LIN {X 0,Y 291.384,Z 318.187,A -85,B 0,C 180,E1 -16597.255,E2 -16597.255} C_VEL
LIN {X 0,Y 291.337,Z 318.196,A -85,B 0,C 180,E1 -16600.642,E2 -16600.642} C_VEL
LIN {X 0,Y 291.402,Z 318.333,A -85,B 0,C 180,E1 -16602.352,E2 -16602.352} C_VEL
LIN {X 0,Y 292.391,Z 323.725,A -85,B 0,C 180,E1 -16606.145,E2 -16606.145} C_VEL
LIN {X 0,Y 293.452,Z 329.609,A -85,B 0,C 180,E1 -16610.03,E2 -16610.03} C_VEL
LIN {X 0,Y 293.964,Z 332.856,A -85,B 0,C 180,E1 -16612.088,E2 -16612.088} C_VEL
LIN {X 0,Y 294.034,Z 334.839,A -85,B 0,C 180,E1 -16613.305,E2 -16613.305} C_VEL
LIN {X 0,Y 293.395,Z 338.972,A -85,B 0,C 180,E1 -16615.742,E2 -16615.742} C_VEL
LIN {X 0,Y 292.231,Z 346.349,A -85,B 0,C 180,E1 -16619.972,E2 -16619.972} C_VEL
LIN {X 0,Y 291.163,Z 353.918,A -85,B 0,C 180,E1 -16624.248,E2 -16624.248} C_VEL
LIN {X 0,Y 290.715,Z 358.235,A -85,B 0,C 180,E1 -16626.649,E2 -16626.649} C_VEL
LIN {X 0,Y 292.536,Z 371.557,A -85,B 0,C 180,E1 -16627.394,E2 -16627.394} C_VEL
LIN {X 0,Y 293.951,Z 383.978,A -85,B 0,C 180,E1 -16628.327,E2 -16628.327} C_VEL
LIN {X 0,Y 294.913,Z 395.491,A -85,B 0,C 180,E1 -16629.421,E2 -16629.421} C_VEL
LIN {X 0,Y 295.433,Z 406.744,A -85,B 0,C 180,E1 -16630.727,E2 -16630.727} C_VEL
LIN {X 0,Y 294.037,Z 417.883,A -85,B 0,C 180,E1 -16632.257,E2 -16632.257} C_VEL
LIN {X 0,Y 292.817,Z 426.678,A -85,B 0,C 180,E1 -16633.752,E2 -16633.752} C_VEL
LIN {X 0,Y 291.678,Z 435.982,A -85,B 0,C 180,E1 -16635.701,E2 -16635.701} C_VEL
LIN {X 0,Y 290.738,Z 444.013,A -85,B 0,C 180,E1 -16637.789,E2 -16637.789} C_VEL
LIN {X 0,Y 290.233,Z 449.451,A -85,B 0,C 180,E1 -16639.536,E2 -16639.536} C_VEL
LIN {X 0,Y 289.879,Z 454.755,A -85,B 0,C 180,E1 -16641.636,E2 -16641.636} C_VEL
LIN {X 0,Y 289.804,Z 459.093,A -85,B 0,C 180,E1 -16643.875,E2 -16643.875} C_VEL
LIN {X 0,Y 289.76,Z 461.832,A -85,B 0,C 180,E1 -16645.827,E2 -16645.827} C_VEL
LIN {X 0,Y 289.832,Z 463.266,A -85,B 0,C 180,E1 -16647.22,E2 -16647.22} C_VEL
LIN {X 0,Y 290.028,Z 464.247,A -85,B 0,C 180,E1 -16648.611,E2 -16648.611} C_VEL
LIN {X 0,Y 290.042,Z 464.802,A -85,B 0,C 180,E1 -16650,E2 -16650} C_VEL
LIN {X 0,Y 289.962,Z 464.944,A -85,B 0,C 180,E1 -16651.389,E2 -16651.389} C_VEL
LIN {X 0,Y 289.747,Z 464.648,A -85,B 0,C 180,E1 -16652.781,E2 -16652.781} C_VEL
LIN {X 0,Y 289.673,Z 463.929,A -85,B 0,C 180,E1 -16654.174,E2 -16654.174} C_VEL
LIN {X 0,Y 289.656,Z 461.291,A -85,B 0,C 180,E1 -16656.968,E2 -16656.968} C_VEL
LIN {X 0,Y 289.897,Z 458.175,A -85,B 0,C 180,E1 -16659.067,E2 -16659.067} C_VEL
LIN {X 0,Y 290.384,Z 454.047,A -85,B 0,C 180,E1 -16661.164,E2 -16661.164} C_VEL
LIN {X 0,Y 291.558,Z 447.849,A -85,B 0,C 180,E1 -16663.593,E2 -16663.593} C_VEL
LIN {X 0,Y 292.919,Z 441.128,A -85,B 0,C 180,E1 -16665.66,E2 -16665.66} C_VEL
LIN {X 0,Y 294.474,Z 433.033,A -85,B 0,C 180,E1 -16667.68,E2 -16667.68} C_VEL
LIN {X 0,Y 296.368,Z 424.574,A -85,B 0,C 180,E1 -16669.39,E2 -16669.39} C_VEL
LIN {X 0,Y 298.591,Z 414.589,A -85,B 0,C 180,E1 -16671.035,E2 -16671.035} C_VEL
LIN {X 0,Y 299.453,Z 405.428,A -85,B 0,C 180,E1 -16672.367,E2 -16672.367} C_VEL
LIN {X 0,Y 299.529,Z 394.395,A -85,B 0,C 180,E1 -16673.783,E2 -16673.783} C_VEL
LIN {X 0,Y 298.6,Z 383.187,A -85,B 0,C 180,E1 -16675.066,E2 -16675.066} C_VEL
LIN {X 0,Y 296.529,Z 370.803,A -85,B 0,C 180,E1 -16676.361,E2 -16676.361} C_VEL
LIN {X 0,Y 293.021,Z 357.071,A -85,B 0,C 180,E1 -16677.694,E2 -16677.694} C_VEL
LIN {X 0,Y 291.962,Z 353.125,A -85,B 0,C 180,E1 -16678.074,E2 -16678.074} C_VEL
LIN {X 0,Y 293.008,Z 346.862,A -85,B 0,C 180,E1 -16681.849,E2 -16681.849} C_VEL
LIN {X 0,Y 294.347,Z 340.748,A -85,B 0,C 180,E1 -16685.727,E2 -16685.727} C_VEL
LIN {X 0,Y 294.85,Z 338.347,A -85,B 0,C 180,E1 -16687.329,E2 -16687.329} C_VEL
LIN {X 0,Y 294.381,Z 334.557,A -85,B 0,C 180,E1 -16690.185,E2 -16690.185} C_VEL
LIN {X 0,Y 293.552,Z 329.912,A -85,B 0,C 180,E1 -16694.09,E2 -16694.09} C_VEL
LIN {X 0,Y 292.79,Z 325.8,A -85,B 0,C 180,E1 -16698.083,E2 -16698.083} C_VEL
LIN {X 0,Y 292.287,Z 322.897,A -85,B 0,C 180,E1 -16701.305,E2 -16701.305} C_VEL
LIN {X 0,Y 291.735,Z 320.101,A -85,B 0,C 180,E1 -16704.993,E2 -16704.993} C_VEL
LIN {X 0,Y 291.376,Z 318.246,A -85,B 0,C 180,E1 -16707.951,E2 -16707.951} C_VEL
LIN {X 0,Y 291.386,Z 318.19,A -85,B 0,C 180,E1 -16711.158,E2 -16711.158} C_VEL
LIN {X 0,Y 291.421,Z 318.185,A -85,B 0,C 180,E1 -16714.272,E2 -16714.272} C_VEL
LIN {X 0,Y 291.386,Z 318.187,A -85,B 0,C 180,E1 -16717.3,E2 -16717.3} C_VEL
LIN {X 0,Y 291.463,Z 318.177,A -85,B 0,C 180,E1 -16720.27,E2 -16720.27} C_VEL
LIN {X 0,Y 291.559,Z 318.164,A -85,B 0,C 180,E1 -16724.624,E2 -16724.624} C_VEL
LIN {X 0,Y 291.533,Z 318.167,A -85,B 0,C 180,E1 -16728.88,E2 -16728.88} C_VEL
LIN {X 0,Y 291.667,Z 318.152,A -85,B 0,C 180,E1 -16731.687,E2 -16731.687} C_VEL
LIN {X 0,Y 291.615,Z 318.162,A -85,B 0,C 180,E1 -16734.468,E2 -16734.468} C_VEL
LIN {X 0,Y 291.892,Z 318.126,A -85,B 0,C 180,E1 -16738.62,E2 -16738.62} C_VEL
LIN {X 0,Y 291.893,Z 318.128,A -85,B 0,C 180,E1 -16741.379,E2 -16741.379} C_VEL
LIN {X 0,Y 291.907,Z 319.951,A -85,B 0,C 180,E1 -16745.526,E2 -16745.526} C_VEL
LIN {X 0,Y 292.082,Z 321.378,A -85,B 0,C 180,E1 -16748.301,E2 -16748.301} C_VEL
LIN {X 0,Y 291.958,Z 322.586,A -85,B 0,C 180,E1 -16750.134,E2 -16750.134} C_VEL
LIN {X 0,Y 293.139,Z 325.506,A -85,B 0,C 180,E1 -16750.48,E2 -16750.48} C_VEL
LIN {X 0,Y 296.261,Z 331.803,A -85,B 0,C 180,E1 -16751.329,E2 -16751.329} C_VEL
LIN {X 0,Y 300.206,Z 341.684,A -85,B 0,C 180,E1 -16752.657,E2 -16752.657} C_VEL
LIN {X 0,Y 303.281,Z 352.214,A -85,B 0,C 180,E1 -16754.103,E2 -16754.103} C_VEL
LIN {X 0,Y 304.6,Z 358.809,A -85,B 0,C 180,E1 -16755.044,E2 -16755.044} C_VEL
LIN {X 0,Y 302.617,Z 370.426,A -85,B 0,C 180,E1 -16756.462,E2 -16756.462} C_VEL
LIN {X 0,Y 300.635,Z 380.69,A -85,B 0,C 180,E1 -16758.044,E2 -16758.044} C_VEL
LIN {X 0,Y 298.697,Z 389.576,A -85,B 0,C 180,E1 -16759.752,E2 -16759.752} C_VEL
LIN {X 0,Y 296.547,Z 398.595,A -85,B 0,C 180,E1 -16761.91,E2 -16761.91} C_VEL
LIN {X 0,Y 294.907,Z 405.165,A -85,B 0,C 180,E1 -16763.899,E2 -16763.899} C_VEL
LIN {X 0,Y 293.27,Z 411.348,A -85,B 0,C 180,E1 -16766.317,E2 -16766.317} C_VEL
LIN {X 0,Y 292.017,Z 416.012,A -85,B 0,C 180,E1 -16768.773,E2 -16768.773} C_VEL
LIN {X 0,Y 291.311,Z 418.312,A -85,B 0,C 180,E1 -16770.44,E2 -16770.44} C_VEL
LIN {X 0,Y 290.723,Z 420.115,A -85,B 0,C 180,E1 -16772.21,E2 -16772.21} C_VEL
LIN {X 0,Y 290.166,Z 421.443,A -85,B 0,C 180,E1 -16774.563,E2 -16774.563} C_VEL
LIN {X 0,Y 289.816,Z 421.556,A -85,B 0,C 180,E1 -16777.319,E2 -16777.319} C_VEL
LIN {X 0,Y 289.773,Z 420.803,A -85,B 0,C 180,E1 -16779.094,E2 -16779.094} C_VEL
LIN {X 0,Y 289.911,Z 418.967,A -85,B 0,C 180,E1 -16781.279,E2 -16781.279} C_VEL
LIN {X 0,Y 290.27,Z 416.159,A -85,B 0,C 180,E1 -16783.418,E2 -16783.418} C_VEL
LIN {X 0,Y 290.82,Z 411.521,A -85,B 0,C 180,E1 -16785.913,E2 -16785.913} C_VEL
LIN {X 0,Y 291.592,Z 405.427,A -85,B 0,C 180,E1 -16788.346,E2 -16788.346} C_VEL
LIN {X 0,Y 292.521,Z 398.224,A -85,B 0,C 180,E1 -16790.564,E2 -16790.564} C_VEL
LIN {X 0,Y 293.568,Z 390.435,A -85,B 0,C 180,E1 -16792.494,E2 -16792.494} C_VEL
LIN {X 0,Y 294.849,Z 381.177,A -85,B 0,C 180,E1 -16794.356,E2 -16794.356} C_VEL
LIN {X 0,Y 296.27,Z 370.145,A -85,B 0,C 180,E1 -16796.125,E2 -16796.125} C_VEL
LIN {X 0,Y 297.43,Z 359.208,A -85,B 0,C 180,E1 -16797.539,E2 -16797.539} C_VEL
LIN {X 0,Y 298.285,Z 349.136,A -85,B 0,C 180,E1 -16798.589,E2 -16798.589} C_VEL
LIN {X 0,Y 295.879,Z 337.582,A -85,B 0,C 180,E1 -16799.734,E2 -16799.734} C_VEL
LIN {X 0,Y 292.465,Z 324.071,A -85,B 0,C 180,E1 -16800.819,E2 -16800.819} C_VEL
LIN {X 0,Y 290.677,Z 318.279,A -85,B 0,C 180,E1 -16801.23,E2 -16801.23} C_VEL
LIN {X 0,Y 291.025,Z 318.232,A -85,B 0,C 180,E1 -16804.235,E2 -16804.235} C_VEL
LIN {X 0,Y 291.29,Z 318.203,A -85,B 0,C 180,E1 -16807.292,E2 -16807.292} C_VEL
LIN {X 0,Y 291.385,Z 318.187,A -85,B 0,C 180,E1 -16810.265,E2 -16810.265} C_VEL
LIN {X 0,Y 291.498,Z 318.174,A -85,B 0,C 180,E1 -16814.665,E2 -16814.665} C_VEL
LIN {X 0,Y 291.536,Z 318.172,A -85,B 0,C 180,E1 -16818.88,E2 -16818.88} C_VEL
LIN {X 0,Y 291.655,Z 318.154,A -85,B 0,C 180,E1 -16821.687,E2 -16821.687} C_VEL
LIN {X 0,Y 291.612,Z 318.159,A -85,B 0,C 180,E1 -16824.468,E2 -16824.468} C_VEL
LIN {X 0,Y 291.89,Z 318.127,A -85,B 0,C 180,E1 -16828.62,E2 -16828.62} C_VEL
LIN {X 0,Y 291.889,Z 318.123,A -85,B 0,C 180,E1 -16831.38,E2 -16831.38} C_VEL
LIN {X 0,Y 291.613,Z 318.158,A -85,B 0,C 180,E1 -16835.532,E2 -16835.532} C_VEL
LIN {X 0,Y 291.669,Z 318.153,A -85,B 0,C 180,E1 -16838.913,E2 -16838.913} C_VEL
LIN {X 0,Y 291.521,Z 318.174,A -85,B 0,C 180,E1 -16842.531,E2 -16842.531} C_VEL
LIN {X 0,Y 291.556,Z 318.164,A -85,B 0,C 180,E1 -16845.376,E2 -16845.376} C_VEL
LIN {X 0,Y 291.451,Z 318.179,A -85,B 0,C 180,E1 -16849.875,E2 -16849.875} C_VEL
LIN {X 0,Y 291.401,Z 318.188,A -85,B 0,C 180,E1 -16854.205,E2 -16854.205} C_VEL
LIN {X 0,Y 291.424,Z 318.181,A -85,B 0,C 180,E1 -16857.272,E2 -16857.272} C_VEL
LIN {X 0,Y 291.338,Z 318.194,A -85,B 0,C 180,E1 -16860.437,E2 -16860.437} C_VEL
LIN {X 0,Y 291.346,Z 318.193,A -85,B 0,C 180,E1 -16863.699,E2 -16863.699} C_VEL
LIN {X 0,Y 291.385,Z 318.186,A -85,B 0,C 180,E1 -16867.256,E2 -16867.256} C_VEL
LIN {X 0,Y 291.335,Z 318.193,A -85,B 0,C 180,E1 -16870.643,E2 -16870.643} C_VEL
LIN {X 0,Y 291.291,Z 318.198,A -85,B 0,C 180,E1 -16874.402,E2 -16874.402} C_VEL
LIN {X 0,Y 291.328,Z 318.194,A -85,B 0,C 180,E1 -16878.405,E2 -16878.405} C_VEL
LIN {X 0,Y 291.366,Z 318.19,A -85,B 0,C 180,E1 -16881.16,E2 -16881.16} C_VEL
LIN {X 0,Y 291.363,Z 318.188,A -85,B 0,C 180,E1 -16884.626,E2 -16884.626} C_VEL
LIN {X 0,Y 291.374,Z 318.189,A -85,B 0,C 180,E1 -16887.951,E2 -16887.951} C_VEL
LIN {X 0,Y 291.388,Z 318.188,A -85,B 0,C 180,E1 -16891.159,E2 -16891.159} C_VEL
LIN {X 0,Y 291.422,Z 318.181,A -85,B 0,C 180,E1 -16894.273,E2 -16894.273} C_VEL
LIN {X 0,Y 291.375,Z 318.192,A -85,B 0,C 180,E1 -16897.299,E2 -16897.299} C_VEL
LIN {X 0,Y 291.442,Z 318.178,A -85,B 0,C 180,E1 -16900.269,E2 -16900.269} C_VEL
LIN {X 0,Y 291.5,Z 318.173,A -85,B 0,C 180,E1 -16904.665,E2 -16904.665} C_VEL
LIN {X 0,Y 291.533,Z 318.17,A -85,B 0,C 180,E1 -16908.881,E2 -16908.881} C_VEL
LIN {X 0,Y 291.671,Z 318.151,A -85,B 0,C 180,E1 -16911.688,E2 -16911.688} C_VEL
LIN {X 0,Y 291.626,Z 318.157,A -85,B 0,C 180,E1 -16914.468,E2 -16914.468} C_VEL
LIN {X 0,Y 291.89,Z 318.125,A -85,B 0,C 180,E1 -16918.621,E2 -16918.621} C_VEL
LIN {X 0,Y 291.867,Z 318.126,A -85,B 0,C 180,E1 -16921.547,E2 -16921.547} C_VEL
LIN {X 0,Y 291.099,Z 318.226,A -85,B 0,C 180,E1 -16922.696,E2 -16922.696} C_VEL
LIN {X 0,Y 288.184,Z 318.588,A -85,B 0,C 180,E1 -16924.567,E2 -16924.567} C_VEL
LIN {X 0,Y 285.759,Z 318.889,A -85,B 0,C 180,E1 -16926.085,E2 -16926.085} C_VEL
LIN {X 0,Y 284.709,Z 319.019,A -85,B 0,C 180,E1 -16927.262,E2 -16927.262} C_VEL
LIN {X 0,Y 284.616,Z 319.029,A -85,B 0,C 180,E1 -16927.661,E2 -16927.661} C_VEL
LIN {X 0,Y 284.486,Z 319.046,A -85,B 0,C 180,E1 -16931.399,E2 -16931.399} C_VEL
LIN {X 0,Y 284.451,Z 319.05,A -85,B 0,C 180,E1 -16935.508,E2 -16935.508} C_VEL
LIN {X 0,Y 284.371,Z 319.063,A -85,B 0,C 180,E1 -16940.243,E2 -16940.243} C_VEL
LIN {X 0,Y 284.329,Z 319.064,A -85,B 0,C 180,E1 -16943.855,E2 -16943.855} C_VEL
LIN {X 0,Y 284.294,Z 319.068,A -85,B 0,C 180,E1 -16948.015,E2 -16948.015} C_VEL
LIN {X 0,Y 284.29,Z 319.07,A -85,B 0,C 180,E1 -16951.275,E2 -16951.275} C_VEL
LIN {X 0,Y 284.344,Z 319.064,A -85,B 0,C 180,E1 -16955.348,E2 -16955.348} C_VEL
LIN {X 0,Y 284.321,Z 319.071,A -85,B 0,C 180,E1 -16958.168,E2 -16958.168} C_VEL
LIN {X 0,Y 284.352,Z 319.177,A -85,B 0,C 180,E1 -16962.017,E2 -16962.017} C_VEL
LIN {X 0,Y 285.255,Z 324.139,A -85,B 0,C 180,E1 -16965.602,E2 -16965.602} C_VEL
LIN {X 0,Y 286.31,Z 329.908,A -85,B 0,C 180,E1 -16969.549,E2 -16969.549} C_VEL
LIN {X 0,Y 286.927,Z 334.071,A -85,B 0,C 180,E1 -16972.24,E2 -16972.24} C_VEL
LIN {X 0,Y 286.847,Z 336.875,A -85,B 0,C 180,E1 -16973.983,E2 -16973.983} C_VEL
LIN {X 0,Y 285.62,Z 343.702,A -85,B 0,C 180,E1 -16978.06,E2 -16978.06} C_VEL
LIN {X 0,Y 284.599,Z 350.468,A -85,B 0,C 180,E1 -16982.018,E2 -16982.018} C_VEL
LIN {X 0,Y 283.704,Z 357.726,A -85,B 0,C 180,E1 -16986.181,E2 -16986.181} C_VEL
LIN {X 0,Y 285.594,Z 371.626,A -85,B 0,C 180,E1 -16987.005,E2 -16987.005} C_VEL
LIN {X 0,Y 287.068,Z 385.13,A -85,B 0,C 180,E1 -16988.078,E2 -16988.078} C_VEL
LIN {X 0,Y 287.989,Z 397.037,A -85,B 0,C 180,E1 -16989.277,E2 -16989.277} C_VEL
LIN {X 0,Y 288.397,Z 407.882,A -85,B 0,C 180,E1 -16990.608,E2 -16990.608} C_VEL
LIN {X 0,Y 286.951,Z 418.62,A -85,B 0,C 180,E1 -16992.173,E2 -16992.173} C_VEL
LIN {X 0,Y 285.492,Z 428.312,A -85,B 0,C 180,E1 -16993.922,E2 -16993.922} C_VEL
LIN {X 0,Y 284.768,Z 434.847,A -85,B 0,C 180,E1 -16995.347,E2 -16995.347} C_VEL
LIN {X 0,Y 283.767,Z 442.978,A -85,B 0,C 180,E1 -16997.484,E2 -16997.484} C_VEL
LIN {X 0,Y 283.186,Z 448.5,A -85,B 0,C 180,E1 -16999.273,E2 -16999.273} C_VEL
LIN {X 0,Y 282.836,Z 453.891,A -85,B 0,C 180,E1 -17001.426,E2 -17001.426} C_VEL
LIN {X 0,Y 282.723,Z 458.606,A -85,B 0,C 180,E1 -17003.899,E2 -17003.899} C_VEL
LIN {X 0,Y 282.695,Z 461.113,A -85,B 0,C 180,E1 -17005.723,E2 -17005.723} C_VEL
LIN {X 0,Y 282.745,Z 462.6,A -85,B 0,C 180,E1 -17007.15,E2 -17007.15} C_VEL
LIN {X 0,Y 282.966,Z 463.625,A -85,B 0,C 180,E1 -17008.577,E2 -17008.577} C_VEL
LIN {X 0,Y 282.985,Z 464.21,A -85,B 0,C 180,E1 -17010,E2 -17010} C_VEL
LIN {X 0,Y 282.883,Z 464.379,A -85,B 0,C 180,E1 -17011.424,E2 -17011.424} C_VEL
LIN {X 0,Y 282.659,Z 464.133,A -85,B 0,C 180,E1 -17012.85,E2 -17012.85} C_VEL
LIN {X 0,Y 282.58,Z 463.45,A -85,B 0,C 180,E1 -17014.279,E2 -17014.279} C_VEL
LIN {X 0,Y 282.58,Z 460.876,A -85,B 0,C 180,E1 -17017.144,E2 -17017.144} C_VEL
LIN {X 0,Y 282.854,Z 457.839,A -85,B 0,C 180,E1 -17019.294,E2 -17019.294} C_VEL
LIN {X 0,Y 283.368,Z 453.789,A -85,B 0,C 180,E1 -17021.444,E2 -17021.444} C_VEL
LIN {X 0,Y 284.421,Z 448.646,A -85,B 0,C 180,E1 -17023.577,E2 -17023.577} C_VEL
LIN {X 0,Y 285.777,Z 442.264,A -85,B 0,C 180,E1 -17025.695,E2 -17025.695} C_VEL
LIN {X 0,Y 287.383,Z 434.737,A -85,B 0,C 180,E1 -17027.726,E2 -17027.726} C_VEL
LIN {X 0,Y 289.254,Z 426.605,A -85,B 0,C 180,E1 -17029.517,E2 -17029.517} C_VEL
LIN {X 0,Y 291.765,Z 416.103,A -85,B 0,C 180,E1 -17031.367,E2 -17031.367} C_VEL
LIN {X 0,Y 292.691,Z 409.429,A -85,B 0,C 180,E1 -17032.407,E2 -17032.407} C_VEL
LIN {X 0,Y 293.122,Z 399.424,A -85,B 0,C 180,E1 -17033.818,E2 -17033.818} C_VEL
LIN {X 0,Y 292.66,Z 388.197,A -85,B 0,C 180,E1 -17035.23,E2 -17035.23} C_VEL
LIN {X 0,Y 291.003,Z 375.62,A -85,B 0,C 180,E1 -17036.672,E2 -17036.672} C_VEL
LIN {X 0,Y 288.042,Z 362.704,A -85,B 0,C 180,E1 -17038.051,E2 -17038.051} C_VEL
LIN {X 0,Y 285.786,Z 355.242,A -85,B 0,C 180,E1 -17038.832,E2 -17038.832} C_VEL
LIN {X 0,Y 285.183,Z 352.471,A -85,B 0,C 180,E1 -17039.064,E2 -17039.064} C_VEL
LIN {X 0,Y 286.522,Z 345.449,A -85,B 0,C 180,E1 -17043.49,E2 -17043.49} C_VEL
LIN {X 0,Y 287.518,Z 341.303,A -85,B 0,C 180,E1 -17046.231,E2 -17046.231} C_VEL
LIN {X 0,Y 287.848,Z 339.323,A -85,B 0,C 180,E1 -17047.618,E2 -17047.618} C_VEL
LIN {X 0,Y 287.338,Z 335.397,A -85,B 0,C 180,E1 -17050.691,E2 -17050.691} C_VEL
LIN {X 0,Y 286.526,Z 330.884,A -85,B 0,C 180,E1 -17054.657,E2 -17054.657} C_VEL
LIN {X 0,Y 285.842,Z 327.153,A -85,B 0,C 180,E1 -17058.405,E2 -17058.405} C_VEL
LIN {X 0,Y 285.283,Z 324.056,A -85,B 0,C 180,E1 -17062.03,E2 -17062.03} C_VEL
LIN {X 0,Y 284.811,Z 321.631,A -85,B 0,C 180,E1 -17065.42,E2 -17065.42} C_VEL
LIN {X 0,Y 284.398,Z 319.649,A -85,B 0,C 180,E1 -17068.738,E2 -17068.738} C_VEL
LIN {X 0,Y 284.362,Z 319.065,A -85,B 0,C 180,E1 -17070.376,E2 -17070.376} C_VEL
LIN {X 0,Y 284.382,Z 319.062,A -85,B 0,C 180,E1 -17073.587,E2 -17073.587} C_VEL
LIN {X 0,Y 284.371,Z 319.065,A -85,B 0,C 180,E1 -17076.707,E2 -17076.707} C_VEL
LIN {X 0,Y 284.409,Z 319.059,A -85,B 0,C 180,E1 -17081.262,E2 -17081.262} C_VEL
LIN {X 0,Y 284.496,Z 319.043,A -85,B 0,C 180,E1 -17084.459,E2 -17084.459} C_VEL
LIN {X 0,Y 284.487,Z 319.046,A -85,B 0,C 180,E1 -17088.601,E2 -17088.601} C_VEL
LIN {X 0,Y 284.622,Z 319.028,A -85,B 0,C 180,E1 -17091.48,E2 -17091.48} C_VEL
LIN {X 0,Y 284.584,Z 319.038,A -85,B 0,C 180,E1 -17094.331,E2 -17094.331} C_VEL
LIN {X 0,Y 284.858,Z 319.002,A -85,B 0,C 180,E1 -17098.586,E2 -17098.586} C_VEL
LIN {X 0,Y 284.927,Z 318.995,A -85,B 0,C 180,E1 -17100,E2 -17100} C_VEL
LIN {X 0,Y 284.909,Z 320.11,A -85,B 0,C 180,E1 -17102.828,E2 -17102.828} C_VEL
LIN {X 0,Y 285.081,Z 322.113,A -85,B 0,C 180,E1 -17107.08,E2 -17107.08} C_VEL
LIN {X 0,Y 285.12,Z 323.327,A -85,B 0,C 180,E1 -17109.091,E2 -17109.091} C_VEL
LIN {X 0,Y 286.352,Z 326.384,A -85,B 0,C 180,E1 -17109.472,E2 -17109.472} C_VEL
LIN {X 0,Y 290.785,Z 335.509,A -85,B 0,C 180,E1 -17110.809,E2 -17110.809} C_VEL
LIN {X 0,Y 294.557,Z 345.346,A -85,B 0,C 180,E1 -17112.225,E2 -17112.225} C_VEL
LIN {X 0,Y 297.25,Z 355.202,A -85,B 0,C 180,E1 -17113.676,E2 -17113.676} C_VEL
LIN {X 0,Y 298.266,Z 360.785,A -85,B 0,C 180,E1 -17114.526,E2 -17114.526} C_VEL
LIN {X 0,Y 296.127,Z 372.488,A -85,B 0,C 180,E1 -17116.015,E2 -17116.015} C_VEL
LIN {X 0,Y 294.053,Z 382.445,A -85,B 0,C 180,E1 -17117.632,E2 -17117.632} C_VEL
LIN {X 0,Y 292.095,Z 390.89,A -85,B 0,C 180,E1 -17119.319,E2 -17119.319} C_VEL
LIN {X 0,Y 290.022,Z 398.999,A -85,B 0,C 180,E1 -17121.315,E2 -17121.315} C_VEL
LIN {X 0,Y 288.301,Z 405.55,A -85,B 0,C 180,E1 -17123.336,E2 -17123.336} C_VEL
LIN {X 0,Y 286.699,Z 411.232,A -85,B 0,C 180,E1 -17125.564,E2 -17125.564} C_VEL
LIN {X 0,Y 285.381,Z 415.772,A -85,B 0,C 180,E1 -17127.898,E2 -17127.898} C_VEL
LIN {X 0,Y 284.373,Z 418.908,A -85,B 0,C 180,E1 -17130.117,E2 -17130.117} C_VEL
LIN {X 0,Y 283.548,Z 421.149,A -85,B 0,C 180,E1 -17132.571,E2 -17132.571} C_VEL
LIN {X 0,Y 283.009,Z 422.174,A -85,B 0,C 180,E1 -17134.965,E2 -17134.965} C_VEL
LIN {X 0,Y 282.754,Z 422.085,A -85,B 0,C 180,E1 -17137.308,E2 -17137.308} C_VEL
LIN {X 0,Y 282.697,Z 420.967,A -85,B 0,C 180,E1 -17139.585,E2 -17139.585} C_VEL
LIN {X 0,Y 282.933,Z 418.507,A -85,B 0,C 180,E1 -17142.119,E2 -17142.119} C_VEL
LIN {X 0,Y 283.309,Z 415.79,A -85,B 0,C 180,E1 -17143.995,E2 -17143.995} C_VEL
LIN {X 0,Y 283.792,Z 411.794,A -85,B 0,C 180,E1 -17146.099,E2 -17146.099} C_VEL
LIN {X 0,Y 284.561,Z 405.866,A -85,B 0,C 180,E1 -17148.496,E2 -17148.496} C_VEL
LIN {X 0,Y 285.527,Z 398.601,A -85,B 0,C 180,E1 -17150.778,E2 -17150.778} C_VEL
LIN {X 0,Y 286.513,Z 391.504,A -85,B 0,C 180,E1 -17152.585,E2 -17152.585} C_VEL
LIN {X 0,Y 287.858,Z 382.083,A -85,B 0,C 180,E1 -17154.547,E2 -17154.547} C_VEL
LIN {X 0,Y 289.188,Z 372.031,A -85,B 0,C 180,E1 -17156.226,E2 -17156.226} C_VEL
LIN {X 0,Y 290.572,Z 359.905,A -85,B 0,C 180,E1 -17157.852,E2 -17157.852} C_VEL
LIN {X 0,Y 291.451,Z 350.44,A -85,B 0,C 180,E1 -17158.867,E2 -17158.867} C_VEL
LIN {X 0,Y 289.155,Z 339.285,A -85,B 0,C 180,E1 -17160.031,E2 -17160.031} C_VEL
LIN {X 0,Y 285.818,Z 326.127,A -85,B 0,C 180,E1 -17161.147,E2 -17161.147} C_VEL
LIN {X 0,Y 283.685,Z 319.149,A -85,B 0,C 180,E1 -17161.668,E2 -17161.668} C_VEL
LIN {X 0,Y 284.058,Z 319.103,A -85,B 0,C 180,E1 -17165.127,E2 -17165.127} C_VEL
LIN {X 0,Y 284.265,Z 319.074,A -85,B 0,C 180,E1 -17168.232,E2 -17168.232} C_VEL
LIN {X 0,Y 284.331,Z 319.069,A -85,B 0,C 180,E1 -17171.256,E2 -17171.256} C_VEL
LIN {X 0,Y 284.464,Z 319.05,A -85,B 0,C 180,E1 -17175.696,E2 -17175.696} C_VEL
LIN {X 0,Y 284.518,Z 319.043,A -85,B 0,C 180,E1 -17180.043,E2 -17180.043} C_VEL
LIN {X 0,Y 284.648,Z 319.03,A -85,B 0,C 180,E1 -17182.909,E2 -17182.909} C_VEL
LIN {X 0,Y 284.856,Z 319.003,A -85,B 0,C 180,E1 -17188.586,E2 -17188.586} C_VEL
LIN {X 0,Y 284.856,Z 318.999,A -85,B 0,C 180,E1 -17191.414,E2 -17191.414} C_VEL
LIN {X 0,Y 284.581,Z 319.034,A -85,B 0,C 180,E1 -17195.669,E2 -17195.669} C_VEL
LIN {X 0,Y 284.611,Z 319.032,A -85,B 0,C 180,E1 -17198.983,E2 -17198.983} C_VEL
LIN {X 0,Y 284.477,Z 319.048,A -85,B 0,C 180,E1 -17202.847,E2 -17202.847} C_VEL
LIN {X 0,Y 284.488,Z 319.045,A -85,B 0,C 180,E1 -17205.768,E2 -17205.768} C_VEL
LIN {X 0,Y 284.379,Z 319.063,A -85,B 0,C 180,E1 -17210.242,E2 -17210.242} C_VEL
LIN {X 0,Y 284.37,Z 319.061,A -85,B 0,C 180,E1 -17213.876,E2 -17213.876} C_VEL
LIN {X 0,Y 284.398,Z 319.056,A -85,B 0,C 180,E1 -17217.174,E2 -17217.174} C_VEL
LIN {X 0,Y 284.297,Z 319.068,A -85,B 0,C 180,E1 -17221.274,E2 -17221.274} C_VEL
LIN {X 0,Y 284.343,Z 319.064,A -85,B 0,C 180,E1 -17225.349,E2 -17225.349} C_VEL
LIN {X 0,Y 284.321,Z 319.068,A -85,B 0,C 180,E1 -17228.168,E2 -17228.168} C_VEL
LIN {X 0,Y 284.27,Z 319.075,A -85,B 0,C 180,E1 -17232.125,E2 -17232.125} C_VEL
LIN {X 0,Y 284.257,Z 319.075,A -85,B 0,C 180,E1 -17236.19,E2 -17236.19} C_VEL
LIN {X 0,Y 284.308,Z 319.07,A -85,B 0,C 180,E1 -17240.024,E2 -17240.024} C_VEL
LIN {X 0,Y 284.336,Z 319.069,A -85,B 0,C 180,E1 -17243.615,E2 -17243.615} C_VEL
LIN {X 0,Y 284.31,Z 319.069,A -85,B 0,C 180,E1 -17247.19,E2 -17247.19} C_VEL
LIN {X 0,Y 284.361,Z 319.061,A -85,B 0,C 180,E1 -17250.377,E2 -17250.377} C_VEL
LIN {X 0,Y 284.383,Z 319.062,A -85,B 0,C 180,E1 -17253.587,E2 -17253.587} C_VEL
LIN {X 0,Y 284.335,Z 319.065,A -85,B 0,C 180,E1 -17256.704,E2 -17256.704} C_VEL
LIN {X 0,Y 284.379,Z 319.059,A -85,B 0,C 180,E1 -17259.905,E2 -17259.905} C_VEL
LIN {X 0,Y 284.45,Z 319.05,A -85,B 0,C 180,E1 -17264.492,E2 -17264.492} C_VEL
LIN {X 0,Y 284.486,Z 319.046,A -85,B 0,C 180,E1 -17268.602,E2 -17268.602} C_VEL
LIN {X 0,Y 284.626,Z 319.03,A -85,B 0,C 180,E1 -17271.48,E2 -17271.48} C_VEL
LIN {X 0,Y 284.596,Z 319.032,A -85,B 0,C 180,E1 -17274.331,E2 -17274.331} C_VEL
LIN {X 0,Y 284.856,Z 319.001,A -85,B 0,C 180,E1 -17278.586,E2 -17278.586} C_VEL
LIN {X 0,Y 284.842,Z 319.002,A -85,B 0,C 180,E1 -17281.507,E2 -17281.507} C_VEL
LIN {X 0,Y 284.651,Z 319.027,A -85,B 0,C 180,E1 -17287.091,E2 -17287.091} C_VEL
LIN {X 0,Y 284.616,Z 319.029,A -85,B 0,C 180,E1 -17287.661,E2 -17287.661} C_VEL
LIN {X 0,Y 283.908,Z 319.121,A -85,B 0,C 180,E1 -17288.842,E2 -17288.842} C_VEL
LIN {X 0,Y 280.983,Z 319.486,A -85,B 0,C 180,E1 -17290.763,E2 -17290.763} C_VEL
LIN {X 0,Y 278.52,Z 319.791,A -85,B 0,C 180,E1 -17292.324,E2 -17292.324} C_VEL
LIN {X 0,Y 277.471,Z 319.918,A -85,B 0,C 180,E1 -17293.535,E2 -17293.535} C_VEL
LIN {X 0,Y 277.389,Z 319.928,A -85,B 0,C 180,E1 -17293.946,E2 -17293.946} C_VEL
LIN {X 0,Y 277.366,Z 319.934,A -85,B 0,C 180,E1 -17296.184,E2 -17296.184} C_VEL
LIN {X 0,Y 277.316,Z 319.942,A -85,B 0,C 180,E1 -17300.332,E2 -17300.332} C_VEL
LIN {X 0,Y 277.285,Z 319.943,A -85,B 0,C 180,E1 -17304.153,E2 -17304.153} C_VEL
LIN {X 0,Y 277.279,Z 319.938,A -85,B 0,C 180,E1 -17307.486,E2 -17307.486} C_VEL
LIN {X 0,Y 277.25,Z 319.95,A -85,B 0,C 180,E1 -17310.473,E2 -17310.473} C_VEL
LIN {X 0,Y 277.249,Z 319.95,A -85,B 0,C 180,E1 -17313.896,E2 -17313.896} C_VEL
LIN {X 0,Y 277.275,Z 319.945,A -85,B 0,C 180,E1 -17317.469,E2 -17317.469} C_VEL
LIN {X 0,Y 277.284,Z 320.074,A -85,B 0,C 180,E1 -17321.708,E2 -17321.708} C_VEL
LIN {X 0,Y 278.379,Z 325.91,A -85,B 0,C 180,E1 -17326.015,E2 -17326.015} C_VEL
LIN {X 0,Y 279.437,Z 331.759,A -85,B 0,C 180,E1 -17330.108,E2 -17330.108} C_VEL
LIN {X 0,Y 279.925,Z 336.085,A -85,B 0,C 180,E1 -17332.946,E2 -17332.946} C_VEL
LIN {X 0,Y 279.326,Z 340.197,A -85,B 0,C 180,E1 -17335.506,E2 -17335.506} C_VEL
LIN {X 0,Y 277.922,Z 348.378,A -85,B 0,C 180,E1 -17340.455,E2 -17340.455} C_VEL
LIN {X 0,Y 276.791,Z 356.405,A -85,B 0,C 180,E1 -17345.232,E2 -17345.232} C_VEL
LIN {X 0,Y 276.698,Z 357.211,A -85,B 0,C 180,E1 -17345.708,E2 -17345.708} C_VEL
LIN {X 0,Y 278.619,Z 371.622,A -85,B 0,C 180,E1 -17346.591,E2 -17346.591} C_VEL
LIN {X 0,Y 280.071,Z 384.955,A -85,B 0,C 180,E1 -17347.695,E2 -17347.695} C_VEL
LIN {X 0,Y 281.013,Z 397.488,A -85,B 0,C 180,E1 -17349.005,E2 -17349.005} C_VEL
LIN {X 0,Y 281.414,Z 407.589,A -85,B 0,C 180,E1 -17350.297,E2 -17350.297} C_VEL
LIN {X 0,Y 279.992,Z 418.288,A -85,B 0,C 180,E1 -17351.903,E2 -17351.903} C_VEL
LIN {X 0,Y 278.384,Z 428.834,A -85,B 0,C 180,E1 -17353.877,E2 -17353.877} C_VEL
LIN {X 0,Y 277.415,Z 436.671,A -85,B 0,C 180,E1 -17355.7,E2 -17355.7} C_VEL
LIN {X 0,Y 276.497,Z 444.313,A -85,B 0,C 180,E1 -17357.895,E2 -17357.895} C_VEL
LIN {X 0,Y 275.88,Z 451.362,A -85,B 0,C 180,E1 -17360.469,E2 -17360.469} C_VEL
LIN {X 0,Y 275.655,Z 456.005,A -85,B 0,C 180,E1 -17362.676,E2 -17362.676} C_VEL
LIN {X 0,Y 275.659,Z 458.441,A -85,B 0,C 180,E1 -17364.147,E2 -17364.147} C_VEL
LIN {X 0,Y 275.631,Z 460.395,A -85,B 0,C 180,E1 -17365.613,E2 -17365.613} C_VEL
LIN {X 0,Y 275.661,Z 461.916,A -85,B 0,C 180,E1 -17367.077,E2 -17367.077} C_VEL
LIN {X 0,Y 275.885,Z 463.001,A -85,B 0,C 180,E1 -17368.54,E2 -17368.54} C_VEL
LIN {X 0,Y 275.93,Z 463.617,A -85,B 0,C 180,E1 -17370,E2 -17370} C_VEL
LIN {X 0,Y 275.805,Z 463.814,A -85,B 0,C 180,E1 -17371.46,E2 -17371.46} C_VEL
LIN {X 0,Y 275.574,Z 463.601,A -85,B 0,C 180,E1 -17372.924,E2 -17372.924} C_VEL
LIN {X 0,Y 275.436,Z 462.101,A -85,B 0,C 180,E1 -17375.659,E2 -17375.659} C_VEL
LIN {X 0,Y 275.502,Z 460.476,A -85,B 0,C 180,E1 -17377.328,E2 -17377.328} C_VEL
LIN {X 0,Y 275.805,Z 457.508,A -85,B 0,C 180,E1 -17379.534,E2 -17379.534} C_VEL
LIN {X 0,Y 276.366,Z 453.531,A -85,B 0,C 180,E1 -17381.738,E2 -17381.738} C_VEL
LIN {X 0,Y 277.494,Z 448.474,A -85,B 0,C 180,E1 -17383.922,E2 -17383.922} C_VEL
LIN {X 0,Y 279.225,Z 441.208,A -85,B 0,C 180,E1 -17386.404,E2 -17386.404} C_VEL
LIN {X 0,Y 280.967,Z 433.264,A -85,B 0,C 180,E1 -17388.56,E2 -17388.56} C_VEL
LIN {X 0,Y 283.482,Z 423.332,A -85,B 0,C 180,E1 -17390.688,E2 -17390.688} C_VEL
LIN {X 0,Y 285.781,Z 413.388,A -85,B 0,C 180,E1 -17392.407,E2 -17392.407} C_VEL
LIN {X 0,Y 286.6,Z 402.569,A -85,B 0,C 180,E1 -17394.07,E2 -17394.07} C_VEL
LIN {X 0,Y 286.443,Z 391.179,A -85,B 0,C 180,E1 -17395.622,E2 -17395.622} C_VEL
LIN {X 0,Y 285.247,Z 379.546,A -85,B 0,C 180,E1 -17397.056,E2 -17397.056} C_VEL
LIN {X 0,Y 282.435,Z 365.834,A -85,B 0,C 180,E1 -17398.657,E2 -17398.657} C_VEL
LIN {X 0,Y 279.447,Z 355.451,A -85,B 0,C 180,E1 -17399.814,E2 -17399.814} C_VEL
LIN {X 0,Y 278.435,Z 351.656,A -85,B 0,C 180,E1 -17400.233,E2 -17400.233} C_VEL
LIN {X 0,Y 279.66,Z 345.943,A -85,B 0,C 180,E1 -17403.972,E2 -17403.972} C_VEL
LIN {X 0,Y 280.665,Z 341.637,A -85,B 0,C 180,E1 -17406.94,E2 -17406.94} C_VEL
LIN {X 0,Y 280.857,Z 340.438,A -85,B 0,C 180,E1 -17407.813,E2 -17407.813} C_VEL
LIN {X 0,Y 280.296,Z 336.252,A -85,B 0,C 180,E1 -17411.218,E2 -17411.218} C_VEL
LIN {X 0,Y 279.609,Z 332.387,A -85,B 0,C 180,E1 -17414.732,E2 -17414.732} C_VEL
LIN {X 0,Y 278.826,Z 328.197,A -85,B 0,C 180,E1 -17419.128,E2 -17419.128} C_VEL
LIN {X 0,Y 278.291,Z 325.314,A -85,B 0,C 180,E1 -17422.692,E2 -17422.692} C_VEL
LIN {X 0,Y 277.781,Z 322.66,A -85,B 0,C 180,E1 -17426.608,E2 -17426.608} C_VEL
LIN {X 0,Y 277.493,Z 321.052,A -85,B 0,C 180,E1 -17429.566,E2 -17429.566} C_VEL
LIN {X 0,Y 277.329,Z 319.94,A -85,B 0,C 180,E1 -17432.495,E2 -17432.495} C_VEL
LIN {X 0,Y 277.333,Z 319.937,A -85,B 0,C 180,E1 -17436.08,E2 -17436.08} C_VEL
LIN {X 0,Y 277.35,Z 319.937,A -85,B 0,C 180,E1 -17440.766,E2 -17440.766} C_VEL
LIN {X 0,Y 277.439,Z 319.926,A -85,B 0,C 180,E1 -17445.326,E2 -17445.326} C_VEL
LIN {X 0,Y 277.461,Z 319.923,A -85,B 0,C 180,E1 -17449.787,E2 -17449.787} C_VEL
LIN {X 0,Y 277.615,Z 319.903,A -85,B 0,C 180,E1 -17452.728,E2 -17452.728} C_VEL
LIN {X 0,Y 277.7,Z 319.892,A -85,B 0,C 180,E1 -17457.098,E2 -17457.098} C_VEL
LIN {X 0,Y 277.824,Z 319.957,A -85,B 0,C 180,E1 -17458.55,E2 -17458.55} C_VEL
LIN {X 0,Y 277.986,Z 321.009,A -85,B 0,C 180,E1 -17461.449,E2 -17461.449} C_VEL
LIN {X 0,Y 278.033,Z 322.925,A -85,B 0,C 180,E1 -17465.803,E2 -17465.803} C_VEL
LIN {X 0,Y 278.169,Z 324.163,A -85,B 0,C 180,E1 -17467.942,E2 -17467.942} C_VEL
LIN {X 0,Y 279.453,Z 327.112,A -85,B 0,C 180,E1 -17468.36,E2 -17468.36} C_VEL
LIN {X 0,Y 280.589,Z 329.079,A -85,B 0,C 180,E1 -17468.69,E2 -17468.69} C_VEL
LIN {X 0,Y 285.193,Z 338.836,A -85,B 0,C 180,E1 -17470.211,E2 -17470.211} C_VEL
LIN {X 0,Y 288.816,Z 348.778,A -85,B 0,C 180,E1 -17471.759,E2 -17471.759} C_VEL
LIN {X 0,Y 291.134,Z 357.655,A -85,B 0,C 180,E1 -17473.148,E2 -17473.148} C_VEL
LIN {X 0,Y 292.039,Z 362.454,A -85,B 0,C 180,E1 -17473.925,E2 -17473.925} C_VEL
LIN {X 0,Y 289.761,Z 374.048,A -85,B 0,C 180,E1 -17475.474,E2 -17475.474} C_VEL
LIN {X 0,Y 287.681,Z 383.392,A -85,B 0,C 180,E1 -17477.047,E2 -17477.047} C_VEL
LIN {X 0,Y 285.349,Z 392.756,A -85,B 0,C 180,E1 -17478.988,E2 -17478.988} C_VEL
LIN {X 0,Y 283.182,Z 400.808,A -85,B 0,C 180,E1 -17481.091,E2 -17481.091} C_VEL
LIN {X 0,Y 281.019,Z 408.256,A -85,B 0,C 180,E1 -17483.587,E2 -17483.587} C_VEL
LIN {X 0,Y 279.287,Z 413.973,A -85,B 0,C 180,E1 -17486.127,E2 -17486.127} C_VEL
LIN {X 0,Y 277.922,Z 418.185,A -85,B 0,C 180,E1 -17488.716,E2 -17488.716} C_VEL
LIN {X 0,Y 277.181,Z 420.261,A -85,B 0,C 180,E1 -17490.471,E2 -17490.471} C_VEL
LIN {X 0,Y 276.386,Z 422.118,A -85,B 0,C 180,E1 -17492.951,E2 -17492.951} C_VEL
LIN {X 0,Y 275.802,Z 422.827,A -85,B 0,C 180,E1 -17495.88,E2 -17495.88} C_VEL
LIN {X 0,Y 275.64,Z 422.428,A -85,B 0,C 180,E1 -17497.776,E2 -17497.776} C_VEL
LIN {X 0,Y 275.645,Z 421.027,A -85,B 0,C 180,E1 -17500.102,E2 -17500.102} C_VEL
LIN {X 0,Y 275.907,Z 418.645,A -85,B 0,C 180,E1 -17502.379,E2 -17502.379} C_VEL
LIN {X 0,Y 276.329,Z 415.32,A -85,B 0,C 180,E1 -17504.59,E2 -17504.59} C_VEL
LIN {X 0,Y 276.862,Z 411.06,A -85,B 0,C 180,E1 -17506.734,E2 -17506.734} C_VEL
LIN {X 0,Y 277.584,Z 405.775,A -85,B 0,C 180,E1 -17508.831,E2 -17508.831} C_VEL
LIN {X 0,Y 278.456,Z 399.391,A -85,B 0,C 180,E1 -17510.877,E2 -17510.877} C_VEL
LIN {X 0,Y 279.587,Z 391.657,A -85,B 0,C 180,E1 -17512.894,E2 -17512.894} C_VEL
LIN {X 0,Y 280.964,Z 382.278,A -85,B 0,C 180,E1 -17514.878,E2 -17514.878} C_VEL
LIN {X 0,Y 282.314,Z 372.281,A -85,B 0,C 180,E1 -17516.579,E2 -17516.579} C_VEL
LIN {X 0,Y 283.662,Z 360.972,A -85,B 0,C 180,E1 -17518.133,E2 -17518.133} C_VEL
LIN {X 0,Y 284.599,Z 351.586,A -85,B 0,C 180,E1 -17519.175,E2 -17519.175} C_VEL
LIN {X 0,Y 282.351,Z 340.756,A -85,B 0,C 180,E1 -17520.349,E2 -17520.349} C_VEL
LIN {X 0,Y 279.163,Z 328.091,A -85,B 0,C 180,E1 -17521.475,E2 -17521.475} C_VEL
LIN {X 0,Y 276.692,Z 320.018,A -85,B 0,C 180,E1 -17522.086,E2 -17522.086} C_VEL
LIN {X 0,Y 277.106,Z 319.966,A -85,B 0,C 180,E1 -17526.059,E2 -17526.059} C_VEL
LIN {X 0,Y 277.267,Z 319.947,A -85,B 0,C 180,E1 -17529.694,E2 -17529.694} C_VEL
LIN {X 0,Y 277.389,Z 319.93,A -85,B 0,C 180,E1 -17534.318,E2 -17534.318} C_VEL
LIN {X 0,Y 277.434,Z 319.925,A -85,B 0,C 180,E1 -17538.308,E2 -17538.308} C_VEL
LIN {X 0,Y 277.57,Z 319.911,A -85,B 0,C 180,E1 -17541.262,E2 -17541.262} C_VEL
LIN {X 0,Y 277.55,Z 319.91,A -85,B 0,C 180,E1 -17544.187,E2 -17544.187} C_VEL
LIN {X 0,Y 277.822,Z 319.879,A -85,B 0,C 180,E1 -17548.55,E2 -17548.55} C_VEL
LIN {X 0,Y 277.822,Z 319.875,A -85,B 0,C 180,E1 -17551.45,E2 -17551.45} C_VEL
LIN {X 0,Y 277.55,Z 319.91,A -85,B 0,C 180,E1 -17555.813,E2 -17555.813} C_VEL
LIN {X 0,Y 277.561,Z 319.909,A -85,B 0,C 180,E1 -17559.069,E2 -17559.069} C_VEL
LIN {X 0,Y 277.418,Z 319.926,A -85,B 0,C 180,E1 -17563.18,E2 -17563.18} C_VEL
LIN {X 0,Y 277.407,Z 319.93,A -85,B 0,C 180,E1 -17566.182,E2 -17566.182} C_VEL
LIN {X 0,Y 277.346,Z 319.939,A -85,B 0,C 180,E1 -17570.35,E2 -17570.35} C_VEL
LIN {X 0,Y 277.32,Z 319.942,A -85,B 0,C 180,E1 -17574.171,E2 -17574.171} C_VEL
LIN {X 0,Y 277.327,Z 319.938,A -85,B 0,C 180,E1 -17577.506,E2 -17577.506} C_VEL
LIN {X 0,Y 277.273,Z 319.945,A -85,B 0,C 180,E1 -17580.482,E2 -17580.482} C_VEL
LIN {X 0,Y 277.248,Z 319.951,A -85,B 0,C 180,E1 -17583.896,E2 -17583.896} C_VEL
LIN {X 0,Y 277.275,Z 319.945,A -85,B 0,C 180,E1 -17587.469,E2 -17587.469} C_VEL
LIN {X 0,Y 277.211,Z 319.952,A -85,B 0,C 180,E1 -17591.237,E2 -17591.237} C_VEL
LIN {X 0,Y 277.202,Z 319.953,A -85,B 0,C 180,E1 -17595.227,E2 -17595.227} C_VEL
LIN {X 0,Y 277.224,Z 319.953,A -85,B 0,C 180,E1 -17599.512,E2 -17599.512} C_VEL
LIN {X 0,Y 277.274,Z 319.944,A -85,B 0,C 180,E1 -17602.532,E2 -17602.532} C_VEL
LIN {X 0,Y 277.249,Z 319.948,A -85,B 0,C 180,E1 -17606.105,E2 -17606.105} C_VEL
LIN {X 0,Y 277.263,Z 319.95,A -85,B 0,C 180,E1 -17609.539,E2 -17609.539} C_VEL
LIN {X 0,Y 277.364,Z 319.933,A -85,B 0,C 180,E1 -17612.865,E2 -17612.865} C_VEL
LIN {X 0,Y 277.3,Z 319.941,A -85,B 0,C 180,E1 -17616.077,E2 -17616.077} C_VEL
LIN {X 0,Y 277.327,Z 319.938,A -85,B 0,C 180,E1 -17620.765,E2 -17620.765} C_VEL
LIN {X 0,Y 277.413,Z 319.93,A -85,B 0,C 180,E1 -17625.325,E2 -17625.325} C_VEL
LIN {X 0,Y 277.46,Z 319.92,A -85,B 0,C 180,E1 -17629.787,E2 -17629.787} C_VEL
LIN {X 0,Y 277.633,Z 319.902,A -85,B 0,C 180,E1 -17632.729,E2 -17632.729} C_VEL
LIN {X 0,Y 277.822,Z 319.876,A -85,B 0,C 180,E1 -17638.551,E2 -17638.551} C_VEL
LIN {X 0,Y 277.821,Z 319.877,A -85,B 0,C 180,E1 -17641.45,E2 -17641.45} C_VEL
LIN {X 0,Y 277.609,Z 319.903,A -85,B 0,C 180,E1 -17647.272,E2 -17647.272} C_VEL
LIN {X 0,Y 277.461,Z 319.922,A -85,B 0,C 180,E1 -17650.213,E2 -17650.213} C_VEL
LIN {X 0,Y 277.389,Z 319.928,A -85,B 0,C 180,E1 -17653.946,E2 -17653.946} C_VEL
LIN {X 0,Y 276.716,Z 320.016,A -85,B 0,C 180,E1 -17655.157,E2 -17655.157} C_VEL
LIN {X 0,Y 273.815,Z 320.376,A -85,B 0,C 180,E1 -17657.13,E2 -17657.13} C_VEL
LIN {X 0,Y 271.365,Z 320.683,A -85,B 0,C 180,E1 -17658.734,E2 -17658.734} C_VEL
LIN {X 0,Y 270.338,Z 320.809,A -85,B 0,C 180,E1 -17659.978,E2 -17659.978} C_VEL
LIN {X 0,Y 270.267,Z 320.818,A -85,B 0,C 180,E1 -17660.4,E2 -17660.4} C_VEL
LIN {X 0,Y 270.23,Z 320.819,A -85,B 0,C 180,E1 -17664.59,E2 -17664.59} C_VEL
LIN {X 0,Y 270.208,Z 320.82,A -85,B 0,C 180,E1 -17667.916,E2 -17667.916} C_VEL
LIN {X 0,Y 270.176,Z 320.828,A -85,B 0,C 180,E1 -17671.35,E2 -17671.35} C_VEL
LIN {X 0,Y 270.205,Z 320.825,A -85,B 0,C 180,E1 -17674.905,E2 -17674.905} C_VEL
LIN {X 0,Y 270.2,Z 320.827,A -85,B 0,C 180,E1 -17678.71,E2 -17678.71} C_VEL
LIN {X 0,Y 270.21,Z 320.835,A -85,B 0,C 180,E1 -17681.313,E2 -17681.313} C_VEL
LIN {X 0,Y 270.977,Z 324.931,A -85,B 0,C 180,E1 -17684.449,E2 -17684.449} C_VEL
LIN {X 0,Y 271.988,Z 330.542,A -85,B 0,C 180,E1 -17688.534,E2 -17688.534} C_VEL
LIN {X 0,Y 272.788,Z 335.227,A -85,B 0,C 180,E1 -17691.806,E2 -17691.806} C_VEL
LIN {X 0,Y 272.745,Z 338.056,A -85,B 0,C 180,E1 -17693.654,E2 -17693.654} C_VEL
LIN {X 0,Y 271.74,Z 343.525,A -85,B 0,C 180,E1 -17697.103,E2 -17697.103} C_VEL
LIN {X 0,Y 270.621,Z 350.259,A -85,B 0,C 180,E1 -17701.286,E2 -17701.286} C_VEL
LIN {X 0,Y 269.681,Z 356.734,A -85,B 0,C 180,E1 -17705.254,E2 -17705.254} C_VEL
LIN {X 0,Y 271.617,Z 371.261,A -85,B 0,C 180,E1 -17706.157,E2 -17706.157} C_VEL
LIN {X 0,Y 273.04,Z 384.588,A -85,B 0,C 180,E1 -17707.288,E2 -17707.288} C_VEL
LIN {X 0,Y 273.958,Z 396.227,A -85,B 0,C 180,E1 -17708.531,E2 -17708.531} C_VEL
LIN {X 0,Y 274.398,Z 407.253,A -85,B 0,C 180,E1 -17709.967,E2 -17709.967} C_VEL
LIN {X 0,Y 273.038,Z 417.927,A -85,B 0,C 180,E1 -17711.62,E2 -17711.62} C_VEL
LIN {X 0,Y 271.513,Z 427.547,A -85,B 0,C 180,E1 -17713.457,E2 -17713.457} C_VEL
LIN {X 0,Y 270.481,Z 435.51,A -85,B 0,C 180,E1 -17715.325,E2 -17715.325} C_VEL
LIN {X 0,Y 269.52,Z 443.297,A -85,B 0,C 180,E1 -17717.577,E2 -17717.577} C_VEL
LIN {X 0,Y 268.853,Z 450.432,A -85,B 0,C 180,E1 -17720.217,E2 -17720.217} C_VEL
LIN {X 0,Y 268.594,Z 455.154,A -85,B 0,C 180,E1 -17722.482,E2 -17722.482} C_VEL
LIN {X 0,Y 268.581,Z 457.666,A -85,B 0,C 180,E1 -17723.992,E2 -17723.992} C_VEL
LIN {X 0,Y 268.57,Z 459.656,A -85,B 0,C 180,E1 -17725.497,E2 -17725.497} C_VEL
LIN {X 0,Y 268.579,Z 461.209,A -85,B 0,C 180,E1 -17727,E2 -17727} C_VEL
LIN {X 0,Y 268.805,Z 462.353,A -85,B 0,C 180,E1 -17728.502,E2 -17728.502} C_VEL
LIN {X 0,Y 268.874,Z 463.017,A -85,B 0,C 180,E1 -17730,E2 -17730} C_VEL
LIN {X 0,Y 268.712,Z 463.245,A -85,B 0,C 180,E1 -17731.499,E2 -17731.499} C_VEL
LIN {X 0,Y 268.405,Z 462.498,A -85,B 0,C 180,E1 -17734.505,E2 -17734.505} C_VEL
LIN {X 0,Y 268.354,Z 461.493,A -85,B 0,C 180,E1 -17736.013,E2 -17736.013} C_VEL
LIN {X 0,Y 268.629,Z 458.253,A -85,B 0,C 180,E1 -17739.031,E2 -17739.031} C_VEL
LIN {X 0,Y 269.122,Z 454.707,A -85,B 0,C 180,E1 -17741.295,E2 -17741.295} C_VEL
LIN {X 0,Y 270.138,Z 450.128,A -85,B 0,C 180,E1 -17743.541,E2 -17743.541} C_VEL
LIN {X 0,Y 271.798,Z 443.342,A -85,B 0,C 180,E1 -17746.139,E2 -17746.139} C_VEL
LIN {X 0,Y 273.584,Z 436.022,A -85,B 0,C 180,E1 -17748.342,E2 -17748.342} C_VEL
LIN {X 0,Y 275.952,Z 427.067,A -85,B 0,C 180,E1 -17750.499,E2 -17750.499} C_VEL
LIN {X 0,Y 278.634,Z 417.088,A -85,B 0,C 180,E1 -17752.427,E2 -17752.427} C_VEL
LIN {X 0,Y 279.715,Z 409.562,A -85,B 0,C 180,E1 -17753.704,E2 -17753.704} C_VEL
LIN {X 0,Y 280.256,Z 399.627,A -85,B 0,C 180,E1 -17755.234,E2 -17755.234} C_VEL
LIN {X 0,Y 279.911,Z 389.341,A -85,B 0,C 180,E1 -17756.667,E2 -17756.667} C_VEL
LIN {X 0,Y 278.71,Z 378.784,A -85,B 0,C 180,E1 -17758.046,E2 -17758.046} C_VEL
LIN {X 0,Y 276.298,Z 366.688,A -85,B 0,C 180,E1 -17759.537,E2 -17759.537} C_VEL
LIN {X 0,Y 273.959,Z 358.511,A -85,B 0,C 180,E1 -17760.534,E2 -17760.534} C_VEL
LIN {X 0,Y 272.647,Z 354.463,A -85,B 0,C 180,E1 -17761.034,E2 -17761.034} C_VEL
LIN {X 0,Y 271.734,Z 350.972,A -85,B 0,C 180,E1 -17761.405,E2 -17761.405} C_VEL
LIN {X 0,Y 273.158,Z 345.163,A -85,B 0,C 180,E1 -17765.373,E2 -17765.373} C_VEL
LIN {X 0,Y 273.856,Z 341.553,A -85,B 0,C 180,E1 -17768.019,E2 -17768.019} C_VEL
LIN {X 0,Y 273.24,Z 337.126,A -85,B 0,C 180,E1 -17771.762,E2 -17771.762} C_VEL
LIN {X 0,Y 272.817,Z 334.645,A -85,B 0,C 180,E1 -17774.071,E2 -17774.071} C_VEL
LIN {X 0,Y 271.995,Z 330.394,A -85,B 0,C 180,E1 -17778.532,E2 -17778.532} C_VEL
LIN {X 0,Y 271.58,Z 327.868,A -85,B 0,C 180,E1 -17781.605,E2 -17781.605} C_VEL
LIN {X 0,Y 271,Z 324.781,A -85,B 0,C 180,E1 -17786.087,E2 -17786.087} C_VEL
LIN {X 0,Y 270.543,Z 322.489,A -85,B 0,C 180,E1 -17790.424,E2 -17790.424} C_VEL
LIN {X 0,Y 270.321,Z 321.14,A -85,B 0,C 180,E1 -17793.77,E2 -17793.77} C_VEL
LIN {X 0,Y 270.238,Z 320.822,A -85,B 0,C 180,E1 -17797.039,E2 -17797.039} C_VEL
LIN {X 0,Y 270.306,Z 320.811,A -85,B 0,C 180,E1 -17800.245,E2 -17800.245} C_VEL
LIN {X 0,Y 270.407,Z 320.799,A -85,B 0,C 180,E1 -17804.935,E2 -17804.935} C_VEL
LIN {X 0,Y 270.414,Z 320.799,A -85,B 0,C 180,E1 -17809.518,E2 -17809.518} C_VEL
LIN {X 0,Y 270.574,Z 320.782,A -85,B 0,C 180,E1 -17812.538,E2 -17812.538} C_VEL
LIN {X 0,Y 270.683,Z 321.098,A -85,B 0,C 180,E1 -17817.023,E2 -17817.023} C_VEL
LIN {X 0,Y 271.062,Z 321.996,A -85,B 0,C 180,E1 -17820,E2 -17820} C_VEL
LIN {X 0,Y 271.029,Z 323.152,A -85,B 0,C 180,E1 -17822.973,E2 -17822.973} C_VEL
LIN {X 0,Y 271.113,Z 324.792,A -85,B 0,C 180,E1 -17826.652,E2 -17826.652} C_VEL
LIN {X 0,Y 272.364,Z 327.735,A -85,B 0,C 180,E1 -17827.087,E2 -17827.087} C_VEL
LIN {X 0,Y 273.702,Z 329.72,A -85,B 0,C 180,E1 -17827.478,E2 -17827.478} C_VEL
LIN {X 0,Y 278.272,Z 338.998,A -85,B 0,C 180,E1 -17829.082,E2 -17829.082} C_VEL
LIN {X 0,Y 282.3,Z 349.394,A -85,B 0,C 180,E1 -17830.812,E2 -17830.812} C_VEL
LIN {X 0,Y 284.968,Z 359.838,A -85,B 0,C 180,E1 -17832.553,E2 -17832.553} C_VEL
LIN {X 0,Y 285.737,Z 364.905,A -85,B 0,C 180,E1 -17833.401,E2 -17833.401} C_VEL
LIN {X 0,Y 283.542,Z 375.181,A -85,B 0,C 180,E1 -17834.832,E2 -17834.832} C_VEL
LIN {X 0,Y 280.992,Z 385.914,A -85,B 0,C 180,E1 -17836.716,E2 -17836.716} C_VEL
LIN {X 0,Y 278.5,Z 395.119,A -85,B 0,C 180,E1 -17838.769,E2 -17838.769} C_VEL
LIN {X 0,Y 276.321,Z 402.59,A -85,B 0,C 180,E1 -17840.859,E2 -17840.859} C_VEL
LIN {X 0,Y 274.546,Z 408.324,A -85,B 0,C 180,E1 -17842.845,E2 -17842.845} C_VEL
LIN {X 0,Y 273.022,Z 413.087,A -85,B 0,C 180,E1 -17844.901,E2 -17844.901} C_VEL
LIN {X 0,Y 271.294,Z 418.112,A -85,B 0,C 180,E1 -17847.794,E2 -17847.794} C_VEL
LIN {X 0,Y 269.976,Z 421.452,A -85,B 0,C 180,E1 -17850.789,E2 -17850.789} C_VEL
LIN {X 0,Y 269.217,Z 423,A -85,B 0,C 180,E1 -17853.345,E2 -17853.345} C_VEL
LIN {X 0,Y 268.729,Z 423.395,A -85,B 0,C 180,E1 -17855.832,E2 -17855.832} C_VEL
LIN {X 0,Y 268.543,Z 422.719,A -85,B 0,C 180,E1 -17858.267,E2 -17858.267} C_VEL
LIN {X 0,Y 268.626,Z 420.841,A -85,B 0,C 180,E1 -17860.849,E2 -17860.849} C_VEL
LIN {X 0,Y 269.087,Z 417.113,A -85,B 0,C 180,E1 -17863.825,E2 -17863.825} C_VEL
LIN {X 0,Y 269.583,Z 413.329,A -85,B 0,C 180,E1 -17865.967,E2 -17865.967} C_VEL
LIN {X 0,Y 270.363,Z 407.554,A -85,B 0,C 180,E1 -17868.488,E2 -17868.488} C_VEL
LIN {X 0,Y 271.384,Z 400.146,A -85,B 0,C 180,E1 -17870.978,E2 -17870.978} C_VEL
LIN {X 0,Y 272.55,Z 392.355,A -85,B 0,C 180,E1 -17873.07,E2 -17873.07} C_VEL
LIN {X 0,Y 274.01,Z 382.714,A -85,B 0,C 180,E1 -17875.161,E2 -17875.161} C_VEL
LIN {X 0,Y 275.451,Z 372.415,A -85,B 0,C 180,E1 -17876.946,E2 -17876.946} C_VEL
LIN {X 0,Y 276.745,Z 361.984,A -85,B 0,C 180,E1 -17878.414,E2 -17878.414} C_VEL
LIN {X 0,Y 277.65,Z 353.601,A -85,B 0,C 180,E1 -17879.386,E2 -17879.386} C_VEL
LIN {X 0,Y 276.679,Z 347.467,A -85,B 0,C 180,E1 -17880.099,E2 -17880.099} C_VEL
LIN {X 0,Y 274.154,Z 336.081,A -85,B 0,C 180,E1 -17881.271,E2 -17881.271} C_VEL
LIN {X 0,Y 270.583,Z 323.973,A -85,B 0,C 180,E1 -17882.317,E2 -17882.317} C_VEL
LIN {X 0,Y 269.689,Z 320.891,A -85,B 0,C 180,E1 -17882.572,E2 -17882.572} C_VEL
LIN {X 0,Y 270.012,Z 320.851,A -85,B 0,C 180,E1 -17885.643,E2 -17885.643} C_VEL
LIN {X 0,Y 270.237,Z 320.824,A -85,B 0,C 180,E1 -17889.43,E2 -17889.43} C_VEL
LIN {X 0,Y 270.332,Z 320.809,A -85,B 0,C 180,E1 -17894.136,E2 -17894.136} C_VEL
LIN {X 0,Y 270.397,Z 320.802,A -85,B 0,C 180,E1 -17897.999,E2 -17897.999} C_VEL
LIN {X 0,Y 270.528,Z 320.79,A -85,B 0,C 180,E1 -17901.032,E2 -17901.032} C_VEL
LIN {X 0,Y 270.52,Z 320.785,A -85,B 0,C 180,E1 -17904.035,E2 -17904.035} C_VEL
LIN {X 0,Y 270.788,Z 320.755,A -85,B 0,C 180,E1 -17908.513,E2 -17908.513} C_VEL
LIN {X 0,Y 270.787,Z 320.751,A -85,B 0,C 180,E1 -17911.487,E2 -17911.487} C_VEL
LIN {X 0,Y 270.567,Z 320.779,A -85,B 0,C 180,E1 -17917.462,E2 -17917.462} C_VEL
LIN {X 0,Y 270.413,Z 320.803,A -85,B 0,C 180,E1 -17920.482,E2 -17920.482} C_VEL
LIN {X 0,Y 270.404,Z 320.8,A -85,B 0,C 180,E1 -17925.065,E2 -17925.065} C_VEL
LIN {X 0,Y 270.302,Z 320.813,A -85,B 0,C 180,E1 -17929.756,E2 -17929.756} C_VEL
LIN {X 0,Y 270.275,Z 320.818,A -85,B 0,C 180,E1 -17934.586,E2 -17934.586} C_VEL
LIN {X 0,Y 270.273,Z 320.819,A -85,B 0,C 180,E1 -17937.909,E2 -17937.909} C_VEL
LIN {X 0,Y 270.185,Z 320.826,A -85,B 0,C 180,E1 -17941.348,E2 -17941.348} C_VEL
LIN {X 0,Y 270.204,Z 320.825,A -85,B 0,C 180,E1 -17944.905,E2 -17944.905} C_VEL
LIN {X 0,Y 270.223,Z 320.821,A -85,B 0,C 180,E1 -17948.717,E2 -17948.717} C_VEL
LIN {X 0,Y 270.166,Z 320.83,A -85,B 0,C 180,E1 -17953.249,E2 -17953.249} C_VEL
LIN {X 0,Y 270.173,Z 320.829,A -85,B 0,C 180,E1 -17957.442,E2 -17957.442} C_VEL
LIN {X 0,Y 270.208,Z 320.827,A -85,B 0,C 180,E1 -17961.375,E2 -17961.375} C_VEL
LIN {X 0,Y 270.204,Z 320.824,A -85,B 0,C 180,E1 -17965.095,E2 -17965.095} C_VEL
LIN {X 0,Y 270.202,Z 320.827,A -85,B 0,C 180,E1 -17969.131,E2 -17969.131} C_VEL
LIN {X 0,Y 270.268,Z 320.816,A -85,B 0,C 180,E1 -17972.146,E2 -17972.146} C_VEL
LIN {X 0,Y 270.241,Z 320.824,A -85,B 0,C 180,E1 -17975.537,E2 -17975.537} C_VEL
LIN {X 0,Y 270.264,Z 320.816,A -85,B 0,C 180,E1 -17980.242,E2 -17980.242} C_VEL
LIN {X 0,Y 270.38,Z 320.805,A -85,B 0,C 180,E1 -17984.934,E2 -17984.934} C_VEL
LIN {X 0,Y 270.413,Z 320.799,A -85,B 0,C 180,E1 -17989.518,E2 -17989.518} C_VEL
LIN {X 0,Y 270.589,Z 320.778,A -85,B 0,C 180,E1 -17992.538,E2 -17992.538} C_VEL
LIN {X 0,Y 270.788,Z 320.752,A -85,B 0,C 180,E1 -17998.513,E2 -17998.513} C_VEL
LIN {X 0,Y 270.787,Z 320.753,A -85,B 0,C 180,E1 -18001.487,E2 -18001.487} C_VEL
LIN {X 0,Y 270.57,Z 320.779,A -85,B 0,C 180,E1 -18007.463,E2 -18007.463} C_VEL
LIN {X 0,Y 270.413,Z 320.802,A -85,B 0,C 180,E1 -18010.482,E2 -18010.482} C_VEL
LIN {X 0,Y 270.381,Z 320.803,A -85,B 0,C 180,E1 -18015.066,E2 -18015.066} C_VEL
LIN {X 0,Y 270.264,Z 320.817,A -85,B 0,C 180,E1 -18019.759,E2 -18019.759} C_VEL
LIN {X 0,Y 270.267,Z 320.818,A -85,B 0,C 180,E1 -18020.4,E2 -18020.4} C_VEL
LIN {X 0,Y 269.632,Z 320.902,A -85,B 0,C 180,E1 -18021.644,E2 -18021.644} C_VEL
LIN {X 0,Y 266.78,Z 321.257,A -85,B 0,C 180,E1 -18023.671,E2 -18023.671} C_VEL
LIN {X 0,Y 264.323,Z 321.557,A -85,B 0,C 180,E1 -18025.318,E2 -18025.318} C_VEL
LIN {X 0,Y 263.246,Z 321.687,A -85,B 0,C 180,E1 -18026.596,E2 -18026.596} C_VEL
LIN {X 0,Y 263.148,Z 321.697,A -85,B 0,C 180,E1 -18027.03,E2 -18027.03} C_VEL
LIN {X 0,Y 263.132,Z 321.705,A -85,B 0,C 180,E1 -18031.274,E2 -18031.274} C_VEL
LIN {X 0,Y 263.176,Z 321.705,A -85,B 0,C 180,E1 -18034.122,E2 -18034.122} C_VEL
LIN {X 0,Y 263.165,Z 321.705,A -85,B 0,C 180,E1 -18037.896,E2 -18037.896} C_VEL
LIN {X 0,Y 263.164,Z 321.708,A -85,B 0,C 180,E1 -18040.987,E2 -18040.987} C_VEL
LIN {X 0,Y 264.08,Z 326.642,A -85,B 0,C 180,E1 -18044.867,E2 -18044.867} C_VEL
LIN {X 0,Y 265.186,Z 332.777,A -85,B 0,C 180,E1 -18049.392,E2 -18049.392} C_VEL
LIN {X 0,Y 265.783,Z 337.172,A -85,B 0,C 180,E1 -18052.493,E2 -18052.493} C_VEL
LIN {X 0,Y 265.238,Z 341.294,A -85,B 0,C 180,E1 -18055.226,E2 -18055.226} C_VEL
LIN {X 0,Y 263.969,Z 348.114,A -85,B 0,C 180,E1 -18059.611,E2 -18059.611} C_VEL
LIN {X 0,Y 262.723,Z 356.111,A -85,B 0,C 180,E1 -18064.658,E2 -18064.658} C_VEL
LIN {X 0,Y 262.703,Z 356.261,A -85,B 0,C 180,E1 -18064.753,E2 -18064.753} C_VEL
LIN {X 0,Y 264.616,Z 370.745,A -85,B 0,C 180,E1 -18065.688,E2 -18065.688} C_VEL
LIN {X 0,Y 266.09,Z 384.686,A -85,B 0,C 180,E1 -18066.916,E2 -18066.916} C_VEL
LIN {X 0,Y 266.915,Z 395.814,A -85,B 0,C 180,E1 -18068.147,E2 -18068.147} C_VEL
LIN {X 0,Y 267.387,Z 406.77,A -85,B 0,C 180,E1 -18069.619,E2 -18069.619} C_VEL
LIN {X 0,Y 266.79,Z 413.006,A -85,B 0,C 180,E1 -18070.575,E2 -18070.575} C_VEL
LIN {X 0,Y 265.103,Z 423.811,A -85,B 0,C 180,E1 -18072.518,E2 -18072.518} C_VEL
LIN {X 0,Y 264.048,Z 431.288,A -85,B 0,C 180,E1 -18074.178,E2 -18074.178} C_VEL
LIN {X 0,Y 263.047,Z 438.473,A -85,B 0,C 180,E1 -18076.086,E2 -18076.086} C_VEL
LIN {X 0,Y 262.117,Z 445.561,A -85,B 0,C 180,E1 -18078.399,E2 -18078.399} C_VEL
LIN {X 0,Y 261.676,Z 451.214,A -85,B 0,C 180,E1 -18080.727,E2 -18080.727} C_VEL
LIN {X 0,Y 261.519,Z 455.626,A -85,B 0,C 180,E1 -18083.054,E2 -18083.054} C_VEL
LIN {X 0,Y 261.509,Z 458.908,A -85,B 0,C 180,E1 -18085.376,E2 -18085.376} C_VEL
LIN {X 0,Y 261.5,Z 460.497,A -85,B 0,C 180,E1 -18086.919,E2 -18086.919} C_VEL
LIN {X 0,Y 261.728,Z 461.682,A -85,B 0,C 180,E1 -18088.461,E2 -18088.461} C_VEL
LIN {X 0,Y 261.819,Z 462.416,A -85,B 0,C 180,E1 -18090,E2 -18090} C_VEL
LIN {X 0,Y 261.619,Z 462.676,A -85,B 0,C 180,E1 -18091.539,E2 -18091.539} C_VEL
LIN {X 0,Y 261.324,Z 461.998,A -85,B 0,C 180,E1 -18094.628,E2 -18094.628} C_VEL
LIN {X 0,Y 261.258,Z 461.062,A -85,B 0,C 180,E1 -18096.177,E2 -18096.177} C_VEL
LIN {X 0,Y 261.563,Z 457.917,A -85,B 0,C 180,E1 -18099.278,E2 -18099.278} C_VEL
LIN {X 0,Y 262.115,Z 454.456,A -85,B 0,C 180,E1 -18101.601,E2 -18101.601} C_VEL
LIN {X 0,Y 263.204,Z 449.964,A -85,B 0,C 180,E1 -18103.905,E2 -18103.905} C_VEL
LIN {X 0,Y 264.981,Z 443.284,A -85,B 0,C 180,E1 -18106.566,E2 -18106.566} C_VEL
LIN {X 0,Y 266.83,Z 436.166,A -85,B 0,C 180,E1 -18108.823,E2 -18108.823} C_VEL
LIN {X 0,Y 269.337,Z 427.402,A -85,B 0,C 180,E1 -18111.026,E2 -18111.026} C_VEL
LIN {X 0,Y 272.353,Z 416.634,A -85,B 0,C 180,E1 -18113.174,E2 -18113.174} C_VEL
LIN {X 0,Y 273.609,Z 406.478,A -85,B 0,C 180,E1 -18114.936,E2 -18114.936} C_VEL
LIN {X 0,Y 273.883,Z 395.256,A -85,B 0,C 180,E1 -18116.683,E2 -18116.683} C_VEL
LIN {X 0,Y 273.088,Z 383.764,A -85,B 0,C 180,E1 -18118.316,E2 -18118.316} C_VEL
LIN {X 0,Y 270.953,Z 370.795,A -85,B 0,C 180,E1 -18120.051,E2 -18120.051} C_VEL
LIN {X 0,Y 267.788,Z 358.822,A -85,B 0,C 180,E1 -18121.628,E2 -18121.628} C_VEL
LIN {X 0,Y 265.968,Z 353.562,A -85,B 0,C 180,E1 -18122.335,E2 -18122.335} C_VEL
LIN {X 0,Y 265.113,Z 350.183,A -85,B 0,C 180,E1 -18122.728,E2 -18122.728} C_VEL
LIN {X 0,Y 266.501,Z 345.059,A -85,B 0,C 180,E1 -18126.396,E2 -18126.396} C_VEL
LIN {X 0,Y 266.85,Z 343.212,A -85,B 0,C 180,E1 -18127.804,E2 -18127.804} C_VEL
LIN {X 0,Y 266.419,Z 339.174,A -85,B 0,C 180,E1 -18131.261,E2 -18131.261} C_VEL
LIN {X 0,Y 265.808,Z 335.844,A -85,B 0,C 180,E1 -18134.448,E2 -18134.448} C_VEL
LIN {X 0,Y 265.105,Z 332.111,A -85,B 0,C 180,E1 -18138.489,E2 -18138.489} C_VEL
LIN {X 0,Y 264.556,Z 329.068,A -85,B 0,C 180,E1 -18142.338,E2 -18142.338} C_VEL
LIN {X 0,Y 264.162,Z 326.604,A -85,B 0,C 180,E1 -18146.034,E2 -18146.034} C_VEL
LIN {X 0,Y 263.735,Z 324.714,A -85,B 0,C 180,E1 -18149.581,E2 -18149.581} C_VEL
LIN {X 0,Y 263.517,Z 323.247,A -85,B 0,C 180,E1 -18153.038,E2 -18153.038} C_VEL
LIN {X 0,Y 263.29,Z 322.22,A -85,B 0,C 180,E1 -18156.397,E2 -18156.397} C_VEL
LIN {X 0,Y 263.267,Z 321.688,A -85,B 0,C 180,E1 -18159.693,E2 -18159.693} C_VEL
LIN {X 0,Y 263.355,Z 321.676,A -85,B 0,C 180,E1 -18164.522,E2 -18164.522} C_VEL
LIN {X 0,Y 263.357,Z 321.676,A -85,B 0,C 180,E1 -18169.233,E2 -18169.233} C_VEL
LIN {X 0,Y 263.537,Z 321.666,A -85,B 0,C 180,E1 -18172.337,E2 -18172.337} C_VEL
LIN {X 0,Y 263.98,Z 323.093,A -85,B 0,C 180,E1 -18178.474,E2 -18178.474} C_VEL
LIN {X 0,Y 264.126,Z 324.1,A -85,B 0,C 180,E1 -18181.525,E2 -18181.525} C_VEL
LIN {X 0,Y 264.116,Z 325.791,A -85,B 0,C 180,E1 -18185.248,E2 -18185.248} C_VEL
LIN {X 0,Y 265.313,Z 328.499,A -85,B 0,C 180,E1 -18185.701,E2 -18185.701} C_VEL
LIN {X 0,Y 266.965,Z 330.832,A -85,B 0,C 180,E1 -18186.227,E2 -18186.227} C_VEL
LIN {X 0,Y 270.928,Z 338.275,A -85,B 0,C 180,E1 -18187.658,E2 -18187.658} C_VEL
LIN {X 0,Y 274.53,Z 346.825,A -85,B 0,C 180,E1 -18189.207,E2 -18189.207} C_VEL
LIN {X 0,Y 277.377,Z 355.479,A -85,B 0,C 180,E1 -18190.754,E2 -18190.754} C_VEL
LIN {X 0,Y 279.277,Z 364.411,A -85,B 0,C 180,E1 -18192.351,E2 -18192.351} C_VEL
LIN {X 0,Y 279.527,Z 366.395,A -85,B 0,C 180,E1 -18192.709,E2 -18192.709} C_VEL
LIN {X 0,Y 277.131,Z 377.289,A -85,B 0,C 180,E1 -18194.315,E2 -18194.315} C_VEL
LIN {X 0,Y 274.857,Z 386.311,A -85,B 0,C 180,E1 -18195.954,E2 -18195.954} C_VEL
LIN {X 0,Y 272.214,Z 395.58,A -85,B 0,C 180,E1 -18198.048,E2 -18198.048} C_VEL
LIN {X 0,Y 269.766,Z 403.457,A -85,B 0,C 180,E1 -18200.3,E2 -18200.3} C_VEL
LIN {X 0,Y 267.942,Z 408.949,A -85,B 0,C 180,E1 -18202.262,E2 -18202.262} C_VEL
LIN {X 0,Y 265.845,Z 414.971,A -85,B 0,C 180,E1 -18205.023,E2 -18205.023} C_VEL
LIN {X 0,Y 264.297,Z 419.108,A -85,B 0,C 180,E1 -18207.654,E2 -18207.654} C_VEL
LIN {X 0,Y 262.999,Z 422.123,A -85,B 0,C 180,E1 -18210.512,E2 -18210.512} C_VEL
LIN {X 0,Y 262.413,Z 423.299,A -85,B 0,C 180,E1 -18212.387,E2 -18212.387} C_VEL
LIN {X 0,Y 261.931,Z 423.902,A -85,B 0,C 180,E1 -18214.295,E2 -18214.295} C_VEL
LIN {X 0,Y 261.61,Z 423.855,A -85,B 0,C 180,E1 -18216.299,E2 -18216.299} C_VEL
LIN {X 0,Y 261.456,Z 422.883,A -85,B 0,C 180,E1 -18218.782,E2 -18218.782} C_VEL
LIN {X 0,Y 261.568,Z 420.924,A -85,B 0,C 180,E1 -18221.207,E2 -18221.207} C_VEL
LIN {X 0,Y 262.075,Z 417.073,A -85,B 0,C 180,E1 -18224.205,E2 -18224.205} C_VEL
LIN {X 0,Y 262.57,Z 413.352,A -85,B 0,C 180,E1 -18226.277,E2 -18226.277} C_VEL
LIN {X 0,Y 263.386,Z 407.416,A -85,B 0,C 180,E1 -18228.855,E2 -18228.855} C_VEL
LIN {X 0,Y 264.539,Z 399.617,A -85,B 0,C 180,E1 -18231.471,E2 -18231.471} C_VEL
LIN {X 0,Y 265.825,Z 391.115,A -85,B 0,C 180,E1 -18233.732,E2 -18233.732} C_VEL
LIN {X 0,Y 267.345,Z 381.301,A -85,B 0,C 180,E1 -18235.812,E2 -18235.812} C_VEL
LIN {X 0,Y 268.852,Z 370.889,A -85,B 0,C 180,E1 -18237.596,E2 -18237.596} C_VEL
LIN {X 0,Y 270.198,Z 359.678,A -85,B 0,C 180,E1 -18239.131,E2 -18239.131} C_VEL
LIN {X 0,Y 270.779,Z 353.808,A -85,B 0,C 180,E1 -18239.809,E2 -18239.809} C_VEL
LIN {X 0,Y 268.31,Z 341.568,A -85,B 0,C 180,E1 -18241.229,E2 -18241.229} C_VEL
LIN {X 0,Y 265.286,Z 330.098,A -85,B 0,C 180,E1 -18242.339,E2 -18242.339} C_VEL
LIN {X 0,Y 262.694,Z 321.764,A -85,B 0,C 180,E1 -18243.055,E2 -18243.055} C_VEL
LIN {X 0,Y 262.987,Z 321.725,A -85,B 0,C 180,E1 -18246.368,E2 -18246.368} C_VEL
LIN {X 0,Y 263.204,Z 321.699,A -85,B 0,C 180,E1 -18249.688,E2 -18249.688} C_VEL
LIN {X 0,Y 263.311,Z 321.685,A -85,B 0,C 180,E1 -18254.519,E2 -18254.519} C_VEL
LIN {X 0,Y 263.355,Z 321.682,A -85,B 0,C 180,E1 -18259.234,E2 -18259.234} C_VEL
LIN {X 0,Y 263.53,Z 321.659,A -85,B 0,C 180,E1 -18262.337,E2 -18262.337} C_VEL
LIN {X 0,Y 263.752,Z 321.631,A -85,B 0,C 180,E1 -18268.473,E2 -18268.473} C_VEL
LIN {X 0,Y 263.752,Z 321.627,A -85,B 0,C 180,E1 -18271.527,E2 -18271.527} C_VEL
LIN {X 0,Y 263.53,Z 321.655,A -85,B 0,C 180,E1 -18277.663,E2 -18277.663} C_VEL
LIN {X 0,Y 263.355,Z 321.681,A -85,B 0,C 180,E1 -18280.766,E2 -18280.766} C_VEL
LIN {X 0,Y 263.352,Z 321.677,A -85,B 0,C 180,E1 -18285.478,E2 -18285.478} C_VEL
LIN {X 0,Y 263.264,Z 321.693,A -85,B 0,C 180,E1 -18290.307,E2 -18290.307} C_VEL
LIN {X 0,Y 263.21,Z 321.696,A -85,B 0,C 180,E1 -18295.291,E2 -18295.291} C_VEL
LIN {X 0,Y 263.181,Z 321.7,A -85,B 0,C 180,E1 -18298.73,E2 -18298.73} C_VEL
LIN {X 0,Y 263.134,Z 321.708,A -85,B 0,C 180,E1 -18302.288,E2 -18302.288} C_VEL
LIN {X 0,Y 263.178,Z 321.704,A -85,B 0,C 180,E1 -18305.98,E2 -18305.98} C_VEL
LIN {X 0,Y 263.116,Z 321.71,A -85,B 0,C 180,E1 -18309.871,E2 -18309.871} C_VEL
LIN {X 0,Y 263.124,Z 321.71,A -85,B 0,C 180,E1 -18313.984,E2 -18313.984} C_VEL
LIN {X 0,Y 263.126,Z 321.707,A -85,B 0,C 180,E1 -18318.407,E2 -18318.407} C_VEL
LIN {X 0,Y 263.187,Z 321.7,A -85,B 0,C 180,E1 -18323.236,E2 -18323.236} C_VEL
LIN {X 0,Y 263.169,Z 321.703,A -85,B 0,C 180,E1 -18325.888,E2 -18325.888} C_VEL
LIN {X 0,Y 263.153,Z 321.708,A -85,B 0,C 180,E1 -18329.507,E2 -18329.507} C_VEL
LIN {X 0,Y 263.196,Z 321.698,A -85,B 0,C 180,E1 -18333.003,E2 -18333.003} C_VEL
LIN {X 0,Y 263.157,Z 321.703,A -85,B 0,C 180,E1 -18336.385,E2 -18336.385} C_VEL
LIN {X 0,Y 263.241,Z 321.693,A -85,B 0,C 180,E1 -18339.692,E2 -18339.692} C_VEL
LIN {X 0,Y 263.326,Z 321.682,A -85,B 0,C 180,E1 -18344.521,E2 -18344.521} C_VEL
LIN {X 0,Y 263.352,Z 321.681,A -85,B 0,C 180,E1 -18349.234,E2 -18349.234} C_VEL
LIN {X 0,Y 263.548,Z 321.654,A -85,B 0,C 180,E1 -18352.338,E2 -18352.338} C_VEL
LIN {X 0,Y 263.753,Z 321.628,A -85,B 0,C 180,E1 -18358.473,E2 -18358.473} C_VEL
LIN {X 0,Y 263.751,Z 321.629,A -85,B 0,C 180,E1 -18361.527,E2 -18361.527} C_VEL
LIN {X 0,Y 263.533,Z 321.655,A -85,B 0,C 180,E1 -18367.663,E2 -18367.663} C_VEL
LIN {X 0,Y 263.356,Z 321.681,A -85,B 0,C 180,E1 -18370.767,E2 -18370.767} C_VEL
LIN {X 0,Y 263.327,Z 321.681,A -85,B 0,C 180,E1 -18375.48,E2 -18375.48} C_VEL
LIN {X 0,Y 263.236,Z 321.696,A -85,B 0,C 180,E1 -18380.371,E2 -18380.371} C_VEL
LIN {X 0,Y 263.174,Z 321.694,A -85,B 0,C 180,E1 -18385.295,E2 -18385.295} C_VEL
LIN {X 0,Y 263.148,Z 321.697,A -85,B 0,C 180,E1 -18387.03,E2 -18387.03} C_VEL
LIN {X 0,Y 262.445,Z 321.789,A -85,B 0,C 180,E1 -18388.308,E2 -18388.308} C_VEL
LIN {X 0,Y 259.566,Z 322.153,A -85,B 0,C 180,E1 -18390.391,E2 -18390.391} C_VEL
LIN {X 0,Y 257.158,Z 322.453,A -85,B 0,C 180,E1 -18392.085,E2 -18392.085} C_VEL
LIN {X 0,Y 256.15,Z 322.576,A -85,B 0,C 180,E1 -18393.4,E2 -18393.4} C_VEL
LIN {X 0,Y 256.081,Z 322.583,A -85,B 0,C 180,E1 -18393.845,E2 -18393.845} C_VEL
LIN {X 0,Y 256.125,Z 322.58,A -85,B 0,C 180,E1 -18397.273,E2 -18397.273} C_VEL
LIN {X 0,Y 256.13,Z 322.716,A -85,B 0,C 180,E1 -18400.799,E2 -18400.799} C_VEL
LIN {X 0,Y 257.034,Z 327.55,A -85,B 0,C 180,E1 -18404.69,E2 -18404.69} C_VEL
LIN {X 0,Y 258.114,Z 333.465,A -85,B 0,C 180,E1 -18409.195,E2 -18409.195} C_VEL
LIN {X 0,Y 258.695,Z 337.305,A -85,B 0,C 180,E1 -18411.985,E2 -18411.985} C_VEL
LIN {X 0,Y 258.54,Z 340.337,A -85,B 0,C 180,E1 -18414.077,E2 -18414.077} C_VEL
LIN {X 0,Y 257.109,Z 347.289,A -85,B 0,C 180,E1 -18418.71,E2 -18418.71} C_VEL
LIN {X 0,Y 255.948,Z 353.933,A -85,B 0,C 180,E1 -18423.059,E2 -18423.059} C_VEL
LIN {X 0,Y 255.696,Z 355.989,A -85,B 0,C 180,E1 -18424.257,E2 -18424.257} C_VEL
LIN {X 0,Y 257.521,Z 369.72,A -85,B 0,C 180,E1 -18425.153,E2 -18425.153} C_VEL
LIN {X 0,Y 258.937,Z 382.714,A -85,B 0,C 180,E1 -18426.313,E2 -18426.313} C_VEL
LIN {X 0,Y 259.896,Z 395.493,A -85,B 0,C 180,E1 -18427.754,E2 -18427.754} C_VEL
LIN {X 0,Y 260.346,Z 406.276,A -85,B 0,C 180,E1 -18429.249,E2 -18429.249} C_VEL
LIN {X 0,Y 260.029,Z 411.379,A -85,B 0,C 180,E1 -18430.048,E2 -18430.048} C_VEL
LIN {X 0,Y 258.457,Z 421.453,A -85,B 0,C 180,E1 -18431.859,E2 -18431.859} C_VEL
LIN {X 0,Y 257.074,Z 430.149,A -85,B 0,C 180,E1 -18433.781,E2 -18433.781} C_VEL
LIN {X 0,Y 255.932,Z 438.641,A -85,B 0,C 180,E1 -18436.097,E2 -18436.097} C_VEL
LIN {X 0,Y 255.022,Z 445.563,A -85,B 0,C 180,E1 -18438.475,E2 -18438.475} C_VEL
LIN {X 0,Y 254.529,Z 451.912,A -85,B 0,C 180,E1 -18441.265,E2 -18441.265} C_VEL
LIN {X 0,Y 254.449,Z 456.404,A -85,B 0,C 180,E1 -18443.901,E2 -18443.901} C_VEL
LIN {X 0,Y 254.449,Z 458.159,A -85,B 0,C 180,E1 -18445.247,E2 -18445.247} C_VEL
LIN {X 0,Y 254.424,Z 459.785,A -85,B 0,C 180,E1 -18446.833,E2 -18446.833} C_VEL
LIN {X 0,Y 254.636,Z 461.004,A -85,B 0,C 180,E1 -18448.418,E2 -18448.418} C_VEL
LIN {X 0,Y 254.764,Z 461.795,A -85,B 0,C 180,E1 -18450,E2 -18450} C_VEL
LIN {X 0,Y 254.527,Z 462.105,A -85,B 0,C 180,E1 -18451.582,E2 -18451.582} C_VEL
LIN {X 0,Y 254.33,Z 461.999,A -85,B 0,C 180,E1 -18453.168,E2 -18453.168} C_VEL
LIN {X 0,Y 254.193,Z 461.124,A -85,B 0,C 180,E1 -18455.531,E2 -18455.531} C_VEL
LIN {X 0,Y 254.289,Z 459.316,A -85,B 0,C 180,E1 -18457.943,E2 -18457.943} C_VEL
LIN {X 0,Y 254.673,Z 456.586,A -85,B 0,C 180,E1 -18460.333,E2 -18460.333} C_VEL
LIN {X 0,Y 255.416,Z 452.871,A -85,B 0,C 180,E1 -18462.717,E2 -18462.717} C_VEL
LIN {X 0,Y 256.791,Z 448.135,A -85,B 0,C 180,E1 -18465.07,E2 -18465.07} C_VEL
LIN {X 0,Y 258.86,Z 441.143,A -85,B 0,C 180,E1 -18467.773,E2 -18467.773} C_VEL
LIN {X 0,Y 260.896,Z 433.621,A -85,B 0,C 180,E1 -18470.088,E2 -18470.088} C_VEL
LIN {X 0,Y 263.743,Z 424.47,A -85,B 0,C 180,E1 -18472.317,E2 -18472.317} C_VEL
LIN {X 0,Y 266.251,Z 415.219,A -85,B 0,C 180,E1 -18474.151,E2 -18474.151} C_VEL
LIN {X 0,Y 267.347,Z 405.505,A -85,B 0,C 180,E1 -18475.903,E2 -18475.903} C_VEL
LIN {X 0,Y 267.599,Z 395.19,A -85,B 0,C 180,E1 -18477.573,E2 -18477.573} C_VEL
LIN {X 0,Y 266.895,Z 384.489,A -85,B 0,C 180,E1 -18479.18,E2 -18479.18} C_VEL
LIN {X 0,Y 264.902,Z 371.703,A -85,B 0,C 180,E1 -18481.013,E2 -18481.013} C_VEL
LIN {X 0,Y 261.313,Z 358.085,A -85,B 0,C 180,E1 -18482.951,E2 -18482.951} C_VEL
LIN {X 0,Y 259.633,Z 353.192,A -85,B 0,C 180,E1 -18483.672,E2 -18483.672} C_VEL
LIN {X 0,Y 258.665,Z 349.9,A -85,B 0,C 180,E1 -18484.097,E2 -18484.097} C_VEL
LIN {X 0,Y 258.637,Z 349.355,A -85,B 0,C 180,E1 -18484.195,E2 -18484.195} C_VEL
LIN {X 0,Y 259.762,Z 345.053,A -85,B 0,C 180,E1 -18487.433,E2 -18487.433} C_VEL
LIN {X 0,Y 259.728,Z 342.618,A -85,B 0,C 180,E1 -18489.486,E2 -18489.486} C_VEL
LIN {X 0,Y 259.151,Z 338.928,A -85,B 0,C 180,E1 -18492.927,E2 -18492.927} C_VEL
LIN {X 0,Y 258.405,Z 334.842,A -85,B 0,C 180,E1 -18497.252,E2 -18497.252} C_VEL
LIN {X 0,Y 257.826,Z 331.66,A -85,B 0,C 180,E1 -18501.174,E2 -18501.174} C_VEL
LIN {X 0,Y 257.365,Z 329.028,A -85,B 0,C 180,E1 -18505.008,E2 -18505.008} C_VEL
LIN {X 0,Y 256.954,Z 326.973,A -85,B 0,C 180,E1 -18508.689,E2 -18508.689} C_VEL
LIN {X 0,Y 256.694,Z 325.376,A -85,B 0,C 180,E1 -18512.261,E2 -18512.261} C_VEL
LIN {X 0,Y 256.469,Z 324.23,A -85,B 0,C 180,E1 -18515.729,E2 -18515.729} C_VEL
LIN {X 0,Y 256.355,Z 323.447,A -85,B 0,C 180,E1 -18519.121,E2 -18519.121} C_VEL
LIN {X 0,Y 256.369,Z 322.883,A -85,B 0,C 180,E1 -18524.089,E2 -18524.089} C_VEL
LIN {X 0,Y 256.37,Z 323.002,A -85,B 0,C 180,E1 -18528.936,E2 -18528.936} C_VEL
LIN {X 0,Y 256.633,Z 323.333,A -85,B 0,C 180,E1 -18532.13,E2 -18532.13} C_VEL
LIN {X 0,Y 257.074,Z 324.684,A -85,B 0,C 180,E1 -18538.433,E2 -18538.433} C_VEL
LIN {X 0,Y 257.213,Z 325.668,A -85,B 0,C 180,E1 -18541.566,E2 -18541.566} C_VEL
LIN {X 0,Y 257.116,Z 326.481,A -85,B 0,C 180,E1 -18543.673,E2 -18543.673} C_VEL
LIN {X 0,Y 258.31,Z 329.384,A -85,B 0,C 180,E1 -18544.193,E2 -18544.193} C_VEL
LIN {X 0,Y 259.979,Z 331.528,A -85,B 0,C 180,E1 -18544.748,E2 -18544.748} C_VEL
LIN {X 0,Y 262.072,Z 335.001,A -85,B 0,C 180,E1 -18545.522,E2 -18545.522} C_VEL
LIN {X 0,Y 266.497,Z 343.922,A -85,B 0,C 180,E1 -18547.364,E2 -18547.364} C_VEL
LIN {X 0,Y 270.079,Z 353.396,A -85,B 0,C 180,E1 -18549.198,E2 -18549.198} C_VEL
LIN {X 0,Y 272.26,Z 361.75,A -85,B 0,C 180,E1 -18550.786,E2 -18550.786} C_VEL
LIN {X 0,Y 273.371,Z 368.328,A -85,B 0,C 180,E1 -18552.047,E2 -18552.047} C_VEL
LIN {X 0,Y 270.915,Z 378.983,A -85,B 0,C 180,E1 -18553.686,E2 -18553.686} C_VEL
LIN {X 0,Y 268.237,Z 388.785,A -85,B 0,C 180,E1 -18555.578,E2 -18555.578} C_VEL
LIN {X 0,Y 265.527,Z 397.452,A -85,B 0,C 180,E1 -18557.662,E2 -18557.662} C_VEL
LIN {X 0,Y 263.065,Z 404.929,A -85,B 0,C 180,E1 -18559.915,E2 -18559.915} C_VEL
LIN {X 0,Y 260.954,Z 410.814,A -85,B 0,C 180,E1 -18562.151,E2 -18562.151} C_VEL
LIN {X 0,Y 258.847,Z 416.306,A -85,B 0,C 180,E1 -18564.888,E2 -18564.888} C_VEL
LIN {X 0,Y 257.214,Z 420.342,A -85,B 0,C 180,E1 -18567.678,E2 -18567.678} C_VEL
LIN {X 0,Y 256.304,Z 422.268,A -85,B 0,C 180,E1 -18569.575,E2 -18569.575} C_VEL
LIN {X 0,Y 255.602,Z 423.636,A -85,B 0,C 180,E1 -18571.528,E2 -18571.528} C_VEL
LIN {X 0,Y 254.888,Z 424.507,A -85,B 0,C 180,E1 -18574.188,E2 -18574.188} C_VEL
LIN {X 0,Y 254.485,Z 424.27,A -85,B 0,C 180,E1 -18576.785,E2 -18576.785} C_VEL
LIN {X 0,Y 254.396,Z 422.903,A -85,B 0,C 180,E1 -18579.45,E2 -18579.45} C_VEL
LIN {X 0,Y 254.7,Z 419.756,A -85,B 0,C 180,E1 -18582.631,E2 -18582.631} C_VEL
LIN {X 0,Y 255.129,Z 416.428,A -85,B 0,C 180,E1 -18584.904,E2 -18584.904} C_VEL
LIN {X 0,Y 255.7,Z 412.153,A -85,B 0,C 180,E1 -18587.155,E2 -18587.155} C_VEL
LIN {X 0,Y 256.487,Z 406.839,A -85,B 0,C 180,E1 -18589.383,E2 -18589.383} C_VEL
LIN {X 0,Y 257.652,Z 399.308,A -85,B 0,C 180,E1 -18591.911,E2 -18591.911} C_VEL
LIN {X 0,Y 259.01,Z 390.553,A -85,B 0,C 180,E1 -18594.231,E2 -18594.231} C_VEL
LIN {X 0,Y 260.637,Z 380.303,A -85,B 0,C 180,E1 -18596.411,E2 -18596.411} C_VEL
LIN {X 0,Y 262.21,Z 369.482,A -85,B 0,C 180,E1 -18598.237,E2 -18598.237} C_VEL
LIN {X 0,Y 263.729,Z 357,A -85,B 0,C 180,E1 -18599.912,E2 -18599.912} C_VEL
LIN {X 0,Y 263.795,Z 354.127,A -85,B 0,C 180,E1 -18600.25,E2 -18600.25} C_VEL
LIN {X 0,Y 261.279,Z 341.916,A -85,B 0,C 180,E1 -18601.7,E2 -18601.7} C_VEL
LIN {X 0,Y 258.59,Z 331.942,A -85,B 0,C 180,E1 -18602.701,E2 -18602.701} C_VEL
LIN {X 0,Y 255.695,Z 322.636,A -85,B 0,C 180,E1 -18603.526,E2 -18603.526} C_VEL
LIN {X 0,Y 255.987,Z 322.6,A -85,B 0,C 180,E1 -18607.396,E2 -18607.396} C_VEL
LIN {X 0,Y 256.127,Z 322.581,A -85,B 0,C 180,E1 -18610.775,E2 -18610.775} C_VEL
LIN {X 0,Y 256.231,Z 322.566,A -85,B 0,C 180,E1 -18614.08,E2 -18614.08} C_VEL
LIN {X 0,Y 256.289,Z 322.562,A -85,B 0,C 180,E1 -18617.327,E2 -18617.327} C_VEL
LIN {X 0,Y 256.435,Z 322.544,A -85,B 0,C 180,E1 -18620.622,E2 -18620.622} C_VEL
LIN {X 0,Y 256.463,Z 322.536,A -85,B 0,C 180,E1 -18623.707,E2 -18623.707} C_VEL
LIN {X 0,Y 256.715,Z 322.508,A -85,B 0,C 180,E1 -18628.431,E2 -18628.431} C_VEL
LIN {X 0,Y 256.715,Z 322.503,A -85,B 0,C 180,E1 -18631.569,E2 -18631.569} C_VEL
LIN {X 0,Y 256.463,Z 322.539,A -85,B 0,C 180,E1 -18636.293,E2 -18636.293} C_VEL
LIN {X 0,Y 256.427,Z 322.541,A -85,B 0,C 180,E1 -18639.465,E2 -18639.465} C_VEL
LIN {X 0,Y 256.257,Z 322.565,A -85,B 0,C 180,E1 -18644.29,E2 -18644.29} C_VEL
LIN {X 0,Y 256.212,Z 322.568,A -85,B 0,C 180,E1 -18647.562,E2 -18647.562} C_VEL
LIN {X 0,Y 256.158,Z 322.573,A -85,B 0,C 180,E1 -18651.12,E2 -18651.12} C_VEL
LIN {X 0,Y 256.19,Z 322.57,A -85,B 0,C 180,E1 -18655.139,E2 -18655.139} C_VEL
LIN {X 0,Y 256.115,Z 322.58,A -85,B 0,C 180,E1 -18659.6,E2 -18659.6} C_VEL
LIN {X 0,Y 256.077,Z 322.585,A -85,B 0,C 180,E1 -18663.292,E2 -18663.292} C_VEL
LIN {X 0,Y 256.124,Z 322.578,A -85,B 0,C 180,E1 -18667.273,E2 -18667.273} C_VEL
LIN {X 0,Y 256.058,Z 322.587,A -85,B 0,C 180,E1 -18671.203,E2 -18671.203} C_VEL
LIN {X 0,Y 256.059,Z 322.589,A -85,B 0,C 180,E1 -18675.53,E2 -18675.53} C_VEL
LIN {X 0,Y 256.056,Z 322.587,A -85,B 0,C 180,E1 -18678.797,E2 -18678.797} C_VEL
LIN {X 0,Y 256.134,Z 322.577,A -85,B 0,C 180,E1 -18682.868,E2 -18682.868} C_VEL
LIN {X 0,Y 256.078,Z 322.584,A -85,B 0,C 180,E1 -18686.709,E2 -18686.709} C_VEL
LIN {X 0,Y 256.141,Z 322.58,A -85,B 0,C 180,E1 -18691.405,E2 -18691.405} C_VEL
LIN {X 0,Y 256.145,Z 322.578,A -85,B 0,C 180,E1 -18695.697,E2 -18695.697} C_VEL
LIN {X 0,Y 256.151,Z 322.578,A -85,B 0,C 180,E1 -18699.104,E2 -18699.104} C_VEL
LIN {X 0,Y 256.261,Z 322.562,A -85,B 0,C 180,E1 -18704.083,E2 -18704.083} C_VEL
LIN {X 0,Y 256.294,Z 322.56,A -85,B 0,C 180,E1 -18708.933,E2 -18708.933} C_VEL
LIN {X 0,Y 256.508,Z 322.531,A -85,B 0,C 180,E1 -18712.126,E2 -18712.126} C_VEL
LIN {X 0,Y 256.498,Z 322.535,A -85,B 0,C 180,E1 -18716.859,E2 -18716.859} C_VEL
LIN {X 0,Y 256.761,Z 322.499,A -85,B 0,C 180,E1 -18720,E2 -18720} C_VEL
LIN {X 0,Y 256.487,Z 322.535,A -85,B 0,C 180,E1 -18723.142,E2 -18723.142} C_VEL
LIN {X 0,Y 256.496,Z 322.532,A -85,B 0,C 180,E1 -18727.875,E2 -18727.875} C_VEL
LIN {X 0,Y 256.298,Z 322.558,A -85,B 0,C 180,E1 -18731.067,E2 -18731.067} C_VEL
LIN {X 0,Y 256.241,Z 322.565,A -85,B 0,C 180,E1 -18734.291,E2 -18734.291} C_VEL
LIN {X 0,Y 256.181,Z 322.572,A -85,B 0,C 180,E1 -18737.564,E2 -18737.564} C_VEL
LIN {X 0,Y 256.145,Z 322.575,A -85,B 0,C 180,E1 -18741.111,E2 -18741.111} C_VEL
LIN {X 0,Y 256.138,Z 322.57,A -85,B 0,C 180,E1 -18745.113,E2 -18745.113} C_VEL
LIN {X 0,Y 256.06,Z 322.584,A -85,B 0,C 180,E1 -18749.607,E2 -18749.607} C_VEL
LIN {X 0,Y 256.081,Z 322.583,A -85,B 0,C 180,E1 -18753.845,E2 -18753.845} C_VEL
LIN {X 0,Y 255.43,Z 322.668,A -85,B 0,C 180,E1 -18754.719,E2 -18754.719} C_VEL
LIN {X 0,Y 252.617,Z 323.024,A -85,B 0,C 180,E1 -18756.091,E2 -18756.091} C_VEL
LIN {X 0,Y 249.74,Z 323.383,A -85,B 0,C 180,E1 -18757.493,E2 -18757.493} C_VEL
LIN {X 0,Y 249.031,Z 323.466,A -85,B 0,C 180,E1 -18758.401,E2 -18758.401} C_VEL
LIN {X 0,Y 249.081,Z 323.565,A -85,B 0,C 180,E1 -18760.464,E2 -18760.464} C_VEL
LIN {X 0,Y 250.011,Z 328.616,A -85,B 0,C 180,E1 -18764.65,E2 -18764.65} C_VEL
LIN {X 0,Y 251.068,Z 334.305,A -85,B 0,C 180,E1 -18769.095,E2 -18769.095} C_VEL
LIN {X 0,Y 251.632,Z 338.305,A -85,B 0,C 180,E1 -18772.087,E2 -18772.087} C_VEL
LIN {X 0,Y 251.412,Z 341.253,A -85,B 0,C 180,E1 -18774.162,E2 -18774.162} C_VEL
LIN {X 0,Y 250.034,Z 347.813,A -85,B 0,C 180,E1 -18778.667,E2 -18778.667} C_VEL
LIN {X 0,Y 248.831,Z 354.439,A -85,B 0,C 180,E1 -18783.134,E2 -18783.134} C_VEL
LIN {X 0,Y 248.717,Z 355.303,A -85,B 0,C 180,E1 -18783.714,E2 -18783.714} C_VEL
LIN {X 0,Y 250.432,Z 368.442,A -85,B 0,C 180,E1 -18784.599,E2 -18784.599} C_VEL
LIN {X 0,Y 251.857,Z 381.597,A -85,B 0,C 180,E1 -18785.786,E2 -18785.786} C_VEL
LIN {X 0,Y 252.853,Z 394.883,A -85,B 0,C 180,E1 -18787.316,E2 -18787.316} C_VEL
LIN {X 0,Y 253.326,Z 405.739,A -85,B 0,C 180,E1 -18788.859,E2 -18788.859} C_VEL
LIN {X 0,Y 253.127,Z 410.883,A -85,B 0,C 180,E1 -18789.692,E2 -18789.692} C_VEL
LIN {X 0,Y 251.402,Z 421.514,A -85,B 0,C 180,E1 -18791.669,E2 -18791.669} C_VEL
LIN {X 0,Y 250.015,Z 430.22,A -85,B 0,C 180,E1 -18793.674,E2 -18793.674} C_VEL
LIN {X 0,Y 248.82,Z 438.726,A -85,B 0,C 180,E1 -18796.108,E2 -18796.108} C_VEL
LIN {X 0,Y 247.926,Z 445.527,A -85,B 0,C 180,E1 -18798.555,E2 -18798.555} C_VEL
LIN {X 0,Y 247.504,Z 450.96,A -85,B 0,C 180,E1 -18801.015,E2 -18801.015} C_VEL
LIN {X 0,Y 247.383,Z 455.802,A -85,B 0,C 180,E1 -18803.899,E2 -18803.899} C_VEL
LIN {X 0,Y 247.393,Z 457.367,A -85,B 0,C 180,E1 -18805.111,E2 -18805.111} C_VEL
LIN {X 0,Y 247.351,Z 459.048,A -85,B 0,C 180,E1 -18806.742,E2 -18806.742} C_VEL
LIN {X 0,Y 247.547,Z 460.308,A -85,B 0,C 180,E1 -18808.373,E2 -18808.373} C_VEL
LIN {X 0,Y 247.708,Z 461.144,A -85,B 0,C 180,E1 -18810,E2 -18810} C_VEL
LIN {X 0,Y 247.437,Z 461.526,A -85,B 0,C 180,E1 -18811.628,E2 -18811.628} C_VEL
LIN {X 0,Y 247.251,Z 461.468,A -85,B 0,C 180,E1 -18813.259,E2 -18813.259} C_VEL
LIN {X 0,Y 247.105,Z 460.775,A -85,B 0,C 180,E1 -18815.465,E2 -18815.465} C_VEL
LIN {X 0,Y 247.212,Z 458.924,A -85,B 0,C 180,E1 -18818.172,E2 -18818.172} C_VEL
LIN {X 0,Y 247.659,Z 456.273,A -85,B 0,C 180,E1 -18820.629,E2 -18820.629} C_VEL
LIN {X 0,Y 248.463,Z 452.665,A -85,B 0,C 180,E1 -18823.079,E2 -18823.079} C_VEL
LIN {X 0,Y 249.914,Z 448.03,A -85,B 0,C 180,E1 -18825.495,E2 -18825.495} C_VEL
LIN {X 0,Y 251.764,Z 442.25,A -85,B 0,C 180,E1 -18827.883,E2 -18827.883} C_VEL
LIN {X 0,Y 253.82,Z 435.184,A -85,B 0,C 180,E1 -18830.25,E2 -18830.25} C_VEL
LIN {X 0,Y 256.659,Z 426.533,A -85,B 0,C 180,E1 -18832.542,E2 -18832.542} C_VEL
LIN {X 0,Y 259.395,Z 417.826,A -85,B 0,C 180,E1 -18834.405,E2 -18834.405} C_VEL
LIN {X 0,Y 260.837,Z 408.315,A -85,B 0,C 180,E1 -18836.244,E2 -18836.244} C_VEL
LIN {X 0,Y 261.382,Z 397.863,A -85,B 0,C 180,E1 -18838.069,E2 -18838.069} C_VEL
LIN {X 0,Y 261.137,Z 389.092,A -85,B 0,C 180,E1 -18839.495,E2 -18839.495} C_VEL
LIN {X 0,Y 259.676,Z 376.665,A -85,B 0,C 180,E1 -18841.41,E2 -18841.41} C_VEL
LIN {X 0,Y 257.249,Z 365.603,A -85,B 0,C 180,E1 -18843.121,E2 -18843.121} C_VEL
LIN {X 0,Y 254.83,Z 357.256,A -85,B 0,C 180,E1 -18844.42,E2 -18844.42} C_VEL
LIN {X 0,Y 253.488,Z 353.079,A -85,B 0,C 180,E1 -18845.06,E2 -18845.06} C_VEL
LIN {X 0,Y 252.334,Z 349.719,A -85,B 0,C 180,E1 -18845.591,E2 -18845.591} C_VEL
LIN {X 0,Y 252.188,Z 348.591,A -85,B 0,C 180,E1 -18845.72,E2 -18845.72} C_VEL
LIN {X 0,Y 252.823,Z 346.086,A -85,B 0,C 180,E1 -18847.703,E2 -18847.703} C_VEL
LIN {X 0,Y 252.726,Z 343.744,A -85,B 0,C 180,E1 -18849.762,E2 -18849.762} C_VEL
LIN {X 0,Y 252.086,Z 339.872,A -85,B 0,C 180,E1 -18853.542,E2 -18853.542} C_VEL
LIN {X 0,Y 251.385,Z 335.979,A -85,B 0,C 180,E1 -18857.858,E2 -18857.858} C_VEL
LIN {X 0,Y 250.837,Z 332.832,A -85,B 0,C 180,E1 -18861.946,E2 -18861.946} C_VEL
LIN {X 0,Y 250.372,Z 330.314,A -85,B 0,C 180,E1 -18865.847,E2 -18865.847} C_VEL
LIN {X 0,Y 249.978,Z 328.363,A -85,B 0,C 180,E1 -18869.598,E2 -18869.598} C_VEL
LIN {X 0,Y 249.758,Z 326.859,A -85,B 0,C 180,E1 -18873.241,E2 -18873.241} C_VEL
LIN {X 0,Y 249.522,Z 325.804,A -85,B 0,C 180,E1 -18876.776,E2 -18876.776} C_VEL
LIN {X 0,Y 249.458,Z 325.096,A -85,B 0,C 180,E1 -18880.24,E2 -18880.24} C_VEL
LIN {X 0,Y 249.492,Z 324.715,A -85,B 0,C 180,E1 -18883.639,E2 -18883.639} C_VEL
LIN {X 0,Y 249.478,Z 324.728,A -85,B 0,C 180,E1 -18888.627,E2 -18888.627} C_VEL
LIN {X 0,Y 249.741,Z 325.01,A -85,B 0,C 180,E1 -18891.911,E2 -18891.911} C_VEL
LIN {X 0,Y 250.152,Z 326.289,A -85,B 0,C 180,E1 -18898.39,E2 -18898.39} C_VEL
LIN {X 0,Y 250.336,Z 326.721,A -85,B 0,C 180,E1 -18900,E2 -18900} C_VEL
LIN {X 0,Y 250.268,Z 327.415,A -85,B 0,C 180,E1 -18901.961,E2 -18901.961} C_VEL
LIN {X 0,Y 251.43,Z 330.23,A -85,B 0,C 180,E1 -18902.503,E2 -18902.503} C_VEL
LIN {X 0,Y 253.235,Z 332.584,A -85,B 0,C 180,E1 -18903.182,E2 -18903.182} C_VEL
LIN {X 0,Y 255.167,Z 335.942,A -85,B 0,C 180,E1 -18903.997,E2 -18903.997} C_VEL
LIN {X 0,Y 259.776,Z 344.255,A -85,B 0,C 180,E1 -18905.963,E2 -18905.963} C_VEL
LIN {X 0,Y 262.995,Z 352.34,A -85,B 0,C 180,E1 -18907.678,E2 -18907.678} C_VEL
LIN {X 0,Y 265.714,Z 361.265,A -85,B 0,C 180,E1 -18909.515,E2 -18909.515} C_VEL
LIN {X 0,Y 267.287,Z 370.363,A -85,B 0,C 180,E1 -18911.373,E2 -18911.373} C_VEL
LIN {X 0,Y 264.682,Z 380.724,A -85,B 0,C 180,E1 -18913.044,E2 -18913.044} C_VEL
LIN {X 0,Y 261.572,Z 391.28,A -85,B 0,C 180,E1 -18915.186,E2 -18915.186} C_VEL
LIN {X 0,Y 258.726,Z 399.826,A -85,B 0,C 180,E1 -18917.385,E2 -18917.385} C_VEL
LIN {X 0,Y 256.015,Z 407.402,A -85,B 0,C 180,E1 -18919.887,E2 -18919.887} C_VEL
LIN {X 0,Y 254.039,Z 412.351,A -85,B 0,C 180,E1 -18921.93,E2 -18921.93} C_VEL
LIN {X 0,Y 251.866,Z 417.633,A -85,B 0,C 180,E1 -18924.743,E2 -18924.743} C_VEL
LIN {X 0,Y 250.174,Z 421.441,A -85,B 0,C 180,E1 -18927.615,E2 -18927.615} C_VEL
LIN {X 0,Y 248.855,Z 423.885,A -85,B 0,C 180,E1 -18930.553,E2 -18930.553} C_VEL
LIN {X 0,Y 248.195,Z 424.814,A -85,B 0,C 180,E1 -18932.548,E2 -18932.548} C_VEL
LIN {X 0,Y 247.728,Z 425.095,A -85,B 0,C 180,E1 -18934.641,E2 -18934.641} C_VEL
LIN {X 0,Y 247.372,Z 424.55,A -85,B 0,C 180,E1 -18937.297,E2 -18937.297} C_VEL
LIN {X 0,Y 247.316,Z 422.994,A -85,B 0,C 180,E1 -18939.891,E2 -18939.891} C_VEL
LIN {X 0,Y 247.662,Z 419.86,A -85,B 0,C 180,E1 -18942.926,E2 -18942.926} C_VEL
LIN {X 0,Y 248.075,Z 416.651,A -85,B 0,C 180,E1 -18945.093,E2 -18945.093} C_VEL
LIN {X 0,Y 248.828,Z 411.331,A -85,B 0,C 180,E1 -18947.852,E2 -18947.852} C_VEL
LIN {X 0,Y 249.888,Z 404.209,A -85,B 0,C 180,E1 -18950.661,E2 -18950.661} C_VEL
LIN {X 0,Y 251.279,Z 395.705,A -85,B 0,C 180,E1 -18953.286,E2 -18953.286} C_VEL
LIN {X 0,Y 252.774,Z 386.69,A -85,B 0,C 180,E1 -18955.493,E2 -18955.493} C_VEL
LIN {X 0,Y 254.277,Z 377.198,A -85,B 0,C 180,E1 -18957.387,E2 -18957.387} C_VEL
LIN {X 0,Y 255.703,Z 367.098,A -85,B 0,C 180,E1 -18959.032,E2 -18959.032} C_VEL
LIN {X 0,Y 256.994,Z 355.803,A -85,B 0,C 180,E1 -18960.511,E2 -18960.511} C_VEL
LIN {X 0,Y 254.579,Z 343.754,A -85,B 0,C 180,E1 -18962.01,E2 -18962.01} C_VEL
LIN {X 0,Y 251.978,Z 334.031,A -85,B 0,C 180,E1 -18963.048,E2 -18963.048} C_VEL
LIN {X 0,Y 248.704,Z 323.505,A -85,B 0,C 180,E1 -18964.021,E2 -18964.021} C_VEL
LIN {X 0,Y 249.042,Z 323.463,A -85,B 0,C 180,E1 -18968.633,E2 -18968.633} C_VEL
LIN {X 0,Y 249.177,Z 323.446,A -85,B 0,C 180,E1 -18973.617,E2 -18973.617} C_VEL
LIN {X 0,Y 249.214,Z 323.445,A -85,B 0,C 180,E1 -18976.961,E2 -18976.961} C_VEL
LIN {X 0,Y 249.437,Z 323.414,A -85,B 0,C 180,E1 -18981.901,E2 -18981.901} C_VEL
LIN {X 0,Y 249.288,Z 323.434,A -85,B 0,C 180,E1 -18985.148,E2 -18985.148} C_VEL
LIN {X 0,Y 249.676,Z 323.384,A -85,B 0,C 180,E1 -18988.387,E2 -18988.387} C_VEL
LIN {X 0,Y 249.676,Z 323.38,A -85,B 0,C 180,E1 -18991.613,E2 -18991.613} C_VEL
LIN {X 0,Y 249.436,Z 323.415,A -85,B 0,C 180,E1 -18996.471,E2 -18996.471} C_VEL
LIN {X 0,Y 249.344,Z 323.423,A -85,B 0,C 180,E1 -18999.736,E2 -18999.736} C_VEL
LIN {X 0,Y 249.207,Z 323.442,A -85,B 0,C 180,E1 -19004.703,E2 -19004.703} C_VEL
LIN {X 0,Y 249.141,Z 323.451,A -85,B 0,C 180,E1 -19008.077,E2 -19008.077} C_VEL
LIN {X 0,Y 249.088,Z 323.454,A -85,B 0,C 180,E1 -19011.518,E2 -19011.518} C_VEL
LIN {X 0,Y 249.132,Z 323.45,A -85,B 0,C 180,E1 -19015.482,E2 -19015.482} C_VEL
LIN {X 0,Y 249.085,Z 323.455,A -85,B 0,C 180,E1 -19018.994,E2 -19018.994} C_VEL
LIN {X 0,Y 249.034,Z 323.464,A -85,B 0,C 180,E1 -19022.426,E2 -19022.426} C_VEL
LIN {X 0,Y 249.065,Z 323.459,A -85,B 0,C 180,E1 -19026.34,E2 -19026.34} C_VEL
LIN {X 0,Y 249.027,Z 323.463,A -85,B 0,C 180,E1 -19030.474,E2 -19030.474} C_VEL
LIN {X 0,Y 249.004,Z 323.465,A -85,B 0,C 180,E1 -19034.879,E2 -19034.879} C_VEL
LIN {X 0,Y 249.017,Z 323.463,A -85,B 0,C 180,E1 -19037.363,E2 -19037.363} C_VEL
LIN {X 0,Y 249.046,Z 323.461,A -85,B 0,C 180,E1 -19042.2,E2 -19042.2} C_VEL
LIN {X 0,Y 249.059,Z 323.461,A -85,B 0,C 180,E1 -19045.642,E2 -19045.642} C_VEL
LIN {X 0,Y 249.054,Z 323.464,A -85,B 0,C 180,E1 -19049.474,E2 -19049.474} C_VEL
LIN {X 0,Y 249.073,Z 323.458,A -85,B 0,C 180,E1 -19053.162,E2 -19053.162} C_VEL
LIN {X 0,Y 249.063,Z 323.459,A -85,B 0,C 180,E1 -19056.731,E2 -19056.731} C_VEL
LIN {X 0,Y 249.088,Z 323.454,A -85,B 0,C 180,E1 -19060.21,E2 -19060.21} C_VEL
LIN {X 0,Y 249.198,Z 323.443,A -85,B 0,C 180,E1 -19063.619,E2 -19063.619} C_VEL
LIN {X 0,Y 249.237,Z 323.437,A -85,B 0,C 180,E1 -19068.616,E2 -19068.616} C_VEL
LIN {X 0,Y 249.45,Z 323.41,A -85,B 0,C 180,E1 -19071.902,E2 -19071.902} C_VEL
LIN {X 0,Y 249.294,Z 323.432,A -85,B 0,C 180,E1 -19075.149,E2 -19075.149} C_VEL
LIN {X 0,Y 249.677,Z 323.381,A -85,B 0,C 180,E1 -19078.387,E2 -19078.387} C_VEL
LIN {X 0,Y 249.674,Z 323.383,A -85,B 0,C 180,E1 -19081.613,E2 -19081.613} C_VEL
LIN {X 0,Y 249.437,Z 323.412,A -85,B 0,C 180,E1 -19086.471,E2 -19086.471} C_VEL
LIN {X 0,Y 249.346,Z 323.423,A -85,B 0,C 180,E1 -19089.737,E2 -19089.737} C_VEL
LIN {X 0,Y 249.186,Z 323.446,A -85,B 0,C 180,E1 -19094.705,E2 -19094.705} C_VEL
LIN {X 0,Y 249.115,Z 323.453,A -85,B 0,C 180,E1 -19098.079,E2 -19098.079} C_VEL
LIN {X 0,Y 249.083,Z 323.454,A -85,B 0,C 180,E1 -19101.519,E2 -19101.519} C_VEL
LIN {X 0,Y 249.09,Z 323.447,A -85,B 0,C 180,E1 -19105.461,E2 -19105.461} C_VEL
LIN {X 0,Y 249.043,Z 323.458,A -85,B 0,C 180,E1 -19108.975,E2 -19108.975} C_VEL
LIN {X 0,Y 249.033,Z 323.466,A -85,B 0,C 180,E1 -19112.426,E2 -19112.426} C_VEL
LIN {X 0,Y 249.066,Z 323.461,A -85,B 0,C 180,E1 -19116.34,E2 -19116.34} C_VEL
LIN {X 0,Y 249.031,Z 323.466,A -85,B 0,C 180,E1 -19118.401,E2 -19118.401} C_VEL
LIN {X 0,Y 248.39,Z 323.894,A -85,B 0,C 180,E1 -19119.747,E2 -19119.747} C_VEL
LIN {X 0,Y 246.988,Z 324.996,A -85,B 0,C 180,E1 -19121.058,E2 -19121.058} C_VEL
LIN {X 0,Y 243.879,Z 328.351,A -85,B 0,C 180,E1 -19123.656,E2 -19123.656} C_VEL
LIN {X 0,Y 243.165,Z 330.125,A -85,B 0,C 180,E1 -19124.992,E2 -19124.992} C_VEL
LIN {X 0,Y 243.181,Z 330.687,A -85,B 0,C 180,E1 -19125.444,E2 -19125.444} C_VEL
LIN {X 0,Y 244.155,Z 335.942,A -85,B 0,C 180,E1 -19129.656,E2 -19129.656} C_VEL
LIN {X 0,Y 244.583,Z 338.91,A -85,B 0,C 180,E1 -19131.925,E2 -19131.925} C_VEL
LIN {X 0,Y 244.47,Z 341.206,A -85,B 0,C 180,E1 -19133.605,E2 -19133.605} C_VEL
LIN {X 0,Y 242.951,Z 348.282,A -85,B 0,C 180,E1 -19138.621,E2 -19138.621} C_VEL
LIN {X 0,Y 241.749,Z 354.796,A -85,B 0,C 180,E1 -19143.136,E2 -19143.136} C_VEL
LIN {X 0,Y 243.696,Z 370.093,A -85,B 0,C 180,E1 -19144.253,E2 -19144.253} C_VEL
LIN {X 0,Y 245.046,Z 383.414,A -85,B 0,C 180,E1 -19145.551,E2 -19145.551} C_VEL
LIN {X 0,Y 245.92,Z 395.877,A -85,B 0,C 180,E1 -19147.084,E2 -19147.084} C_VEL
LIN {X 0,Y 246.347,Z 407.716,A -85,B 0,C 180,E1 -19148.889,E2 -19148.889} C_VEL
LIN {X 0,Y 245.844,Z 412.56,A -85,B 0,C 180,E1 -19149.719,E2 -19149.719} C_VEL
LIN {X 0,Y 244.286,Z 421.863,A -85,B 0,C 180,E1 -19151.551,E2 -19151.551} C_VEL
LIN {X 0,Y 242.916,Z 430.423,A -85,B 0,C 180,E1 -19153.615,E2 -19153.615} C_VEL
LIN {X 0,Y 241.692,Z 438.754,A -85,B 0,C 180,E1 -19156.119,E2 -19156.119} C_VEL
LIN {X 0,Y 240.818,Z 445.453,A -85,B 0,C 180,E1 -19158.639,E2 -19158.639} C_VEL
LIN {X 0,Y 240.352,Z 451.569,A -85,B 0,C 180,E1 -19161.593,E2 -19161.593} C_VEL
LIN {X 0,Y 240.31,Z 455.206,A -85,B 0,C 180,E1 -19163.909,E2 -19163.909} C_VEL
LIN {X 0,Y 240.281,Z 458.31,A -85,B 0,C 180,E1 -19166.646,E2 -19166.646} C_VEL
LIN {X 0,Y 240.458,Z 459.612,A -85,B 0,C 180,E1 -19168.325,E2 -19168.325} C_VEL
LIN {X 0,Y 240.652,Z 460.492,A -85,B 0,C 180,E1 -19170,E2 -19170} C_VEL
LIN {X 0,Y 240.35,Z 460.918,A -85,B 0,C 180,E1 -19171.676,E2 -19171.676} C_VEL
LIN {X 0,Y 240.173,Z 460.935,A -85,B 0,C 180,E1 -19173.355,E2 -19173.355} C_VEL
LIN {X 0,Y 240.026,Z 460.368,A -85,B 0,C 180,E1 -19175.418,E2 -19175.418} C_VEL
LIN {X 0,Y 240.156,Z 458.529,A -85,B 0,C 180,E1 -19178.414,E2 -19178.414} C_VEL
LIN {X 0,Y 240.638,Z 455.97,A -85,B 0,C 180,E1 -19180.943,E2 -19180.943} C_VEL
LIN {X 0,Y 241.528,Z 452.459,A -85,B 0,C 180,E1 -19183.461,E2 -19183.461} C_VEL
LIN {X 0,Y 243.036,Z 447.93,A -85,B 0,C 180,E1 -19185.945,E2 -19185.945} C_VEL
LIN {X 0,Y 245.403,Z 441.08,A -85,B 0,C 180,E1 -19188.873,E2 -19188.873} C_VEL
LIN {X 0,Y 247.624,Z 434.135,A -85,B 0,C 180,E1 -19191.215,E2 -19191.215} C_VEL
LIN {X 0,Y 250.733,Z 425.367,A -85,B 0,C 180,E1 -19193.542,E2 -19193.542} C_VEL
LIN {X 0,Y 253.385,Z 416.576,A -85,B 0,C 180,E1 -19195.462,E2 -19195.462} C_VEL
LIN {X 0,Y 254.881,Z 405.81,A -85,B 0,C 180,E1 -19197.612,E2 -19197.612} C_VEL
LIN {X 0,Y 255.296,Z 395.416,A -85,B 0,C 180,E1 -19199.477,E2 -19199.477} C_VEL
LIN {X 0,Y 254.389,Z 382.428,A -85,B 0,C 180,E1 -19201.663,E2 -19201.663} C_VEL
LIN {X 0,Y 252.637,Z 371.687,A -85,B 0,C 180,E1 -19203.43,E2 -19203.43} C_VEL
LIN {X 0,Y 249.579,Z 359.793,A -85,B 0,C 180,E1 -19205.426,E2 -19205.426} C_VEL
LIN {X 0,Y 248.528,Z 356.386,A -85,B 0,C 180,E1 -19206.02,E2 -19206.02} C_VEL
LIN {X 0,Y 247.3,Z 352.529,A -85,B 0,C 180,E1 -19206.67,E2 -19206.67} C_VEL
LIN {X 0,Y 245.968,Z 349.145,A -85,B 0,C 180,E1 -19207.295,E2 -19207.295} C_VEL
LIN {X 0,Y 245.738,Z 347.703,A -85,B 0,C 180,E1 -19207.504,E2 -19207.504} C_VEL
LIN {X 0,Y 245.8,Z 345.502,A -85,B 0,C 180,E1 -19209.466,E2 -19209.466} C_VEL
LIN {X 0,Y 245.48,Z 342.991,A -85,B 0,C 180,E1 -19211.894,E2 -19211.894} C_VEL
LIN {X 0,Y 244.711,Z 338.828,A -85,B 0,C 180,E1 -19216.427,E2 -19216.427} C_VEL
LIN {X 0,Y 244.075,Z 335.452,A -85,B 0,C 180,E1 -19220.693,E2 -19220.693} C_VEL
LIN {X 0,Y 243.623,Z 332.744,A -85,B 0,C 180,E1 -19224.763,E2 -19224.763} C_VEL
LIN {X 0,Y 243.213,Z 330.625,A -85,B 0,C 180,E1 -19228.658,E2 -19228.658} C_VEL
LIN {X 0,Y 242.952,Z 328.998,A -85,B 0,C 180,E1 -19232.429,E2 -19232.429} C_VEL
LIN {X 0,Y 242.703,Z 327.836,A -85,B 0,C 180,E1 -19236.084,E2 -19236.084} C_VEL
LIN {X 0,Y 242.59,Z 327.043,A -85,B 0,C 180,E1 -19239.656,E2 -19239.656} C_VEL
LIN {X 0,Y 242.594,Z 326.577,A -85,B 0,C 180,E1 -19243.16,E2 -19243.16} C_VEL
LIN {X 0,Y 242.564,Z 326.444,A -85,B 0,C 180,E1 -19246.597,E2 -19246.597} C_VEL
LIN {X 0,Y 242.836,Z 326.709,A -85,B 0,C 180,E1 -19251.679,E2 -19251.679} C_VEL
LIN {X 0,Y 242.987,Z 327.566,A -85,B 0,C 180,E1 -19256.684,E2 -19256.684} C_VEL
LIN {X 0,Y 243.458,Z 328.52,A -85,B 0,C 180,E1 -19260.028,E2 -19260.028} C_VEL
LIN {X 0,Y 244.719,Z 331.354,A -85,B 0,C 180,E1 -19260.679,E2 -19260.679} C_VEL
LIN {X 0,Y 246.507,Z 333.507,A -85,B 0,C 180,E1 -19261.426,E2 -19261.426} C_VEL
LIN {X 0,Y 248.572,Z 337.055,A -85,B 0,C 180,E1 -19262.38,E2 -19262.38} C_VEL
LIN {X 0,Y 253.954,Z 346.856,A -85,B 0,C 180,E1 -19264.941,E2 -19264.941} C_VEL
LIN {X 0,Y 257.011,Z 354.231,A -85,B 0,C 180,E1 -19266.649,E2 -19266.649} C_VEL
LIN {X 0,Y 259.57,Z 362.827,A -85,B 0,C 180,E1 -19268.564,E2 -19268.564} C_VEL
LIN {X 0,Y 261.239,Z 372.461,A -85,B 0,C 180,E1 -19270.658,E2 -19270.658} C_VEL
LIN {X 0,Y 258.212,Z 383.597,A -85,B 0,C 180,E1 -19272.576,E2 -19272.576} C_VEL
LIN {X 0,Y 255.589,Z 391.829,A -85,B 0,C 180,E1 -19274.328,E2 -19274.328} C_VEL
LIN {X 0,Y 252.589,Z 400.299,A -85,B 0,C 180,E1 -19276.544,E2 -19276.544} C_VEL
LIN {X 0,Y 249.898,Z 407.317,A -85,B 0,C 180,E1 -19278.87,E2 -19278.87} C_VEL
LIN {X 0,Y 247.13,Z 413.942,A -85,B 0,C 180,E1 -19281.697,E2 -19281.697} C_VEL
LIN {X 0,Y 244.894,Z 418.929,A -85,B 0,C 180,E1 -19284.589,E2 -19284.589} C_VEL
LIN {X 0,Y 243.128,Z 422.484,A -85,B 0,C 180,E1 -19287.549,E2 -19287.549} C_VEL
LIN {X 0,Y 242.151,Z 424.159,A -85,B 0,C 180,E1 -19289.564,E2 -19289.564} C_VEL
LIN {X 0,Y 241.176,Z 425.434,A -85,B 0,C 180,E1 -19292.319,E2 -19292.319} C_VEL
LIN {X 0,Y 240.557,Z 425.627,A -85,B 0,C 180,E1 -19295.111,E2 -19295.111} C_VEL
LIN {X 0,Y 240.244,Z 424.728,A -85,B 0,C 180,E1 -19297.903,E2 -19297.903} C_VEL
LIN {X 0,Y 240.249,Z 422.92,A -85,B 0,C 180,E1 -19300.484,E2 -19300.484} C_VEL
LIN {X 0,Y 240.606,Z 420.082,A -85,B 0,C 180,E1 -19303.093,E2 -19303.093} C_VEL
LIN {X 0,Y 241.104,Z 416.326,A -85,B 0,C 180,E1 -19305.606,E2 -19305.606} C_VEL
LIN {X 0,Y 241.961,Z 410.676,A -85,B 0,C 180,E1 -19308.455,E2 -19308.455} C_VEL
LIN {X 0,Y 243.084,Z 403.329,A -85,B 0,C 180,E1 -19311.317,E2 -19311.317} C_VEL
LIN {X 0,Y 244.343,Z 395.751,A -85,B 0,C 180,E1 -19313.645,E2 -19313.645} C_VEL
LIN {X 0,Y 245.948,Z 386.409,A -85,B 0,C 180,E1 -19315.963,E2 -19315.963} C_VEL
LIN {X 0,Y 247.467,Z 377.074,A -85,B 0,C 180,E1 -19317.847,E2 -19317.847} C_VEL
LIN {X 0,Y 249,Z 366.357,A -85,B 0,C 180,E1 -19319.598,E2 -19319.598} C_VEL
LIN {X 0,Y 250.047,Z 357.881,A -85,B 0,C 180,E1 -19320.745,E2 -19320.745} C_VEL
LIN {X 0,Y 249.413,Z 353.22,A -85,B 0,C 180,E1 -19321.378,E2 -19321.378} C_VEL
LIN {X 0,Y 247.156,Z 342.495,A -85,B 0,C 180,E1 -19322.708,E2 -19322.708} C_VEL
LIN {X 0,Y 243.684,Z 330.716,A -85,B 0,C 180,E1 -19323.965,E2 -19323.965} C_VEL
LIN {X 0,Y 241.693,Z 324.378,A -85,B 0,C 180,E1 -19324.555,E2 -19324.555} C_VEL
LIN {X 0,Y 241.964,Z 324.344,A -85,B 0,C 180,E1 -19328.351,E2 -19328.351} C_VEL
LIN {X 0,Y 242.116,Z 324.327,A -85,B 0,C 180,E1 -19333.316,E2 -19333.316} C_VEL
LIN {X 0,Y 242.152,Z 324.322,A -85,B 0,C 180,E1 -19336.574,E2 -19336.574} C_VEL
LIN {X 0,Y 242.387,Z 324.293,A -85,B 0,C 180,E1 -19341.664,E2 -19341.664} C_VEL
LIN {X 0,Y 242.248,Z 324.312,A -85,B 0,C 180,E1 -19345.007,E2 -19345.007} C_VEL
LIN {X 0,Y 242.637,Z 324.261,A -85,B 0,C 180,E1 -19348.34,E2 -19348.34} C_VEL
LIN {X 0,Y 242.637,Z 324.257,A -85,B 0,C 180,E1 -19351.66,E2 -19351.66} C_VEL
LIN {X 0,Y 242.407,Z 324.29,A -85,B 0,C 180,E1 -19356.66,E2 -19356.66} C_VEL
LIN {X 0,Y 242.268,Z 324.306,A -85,B 0,C 180,E1 -19360.024,E2 -19360.024} C_VEL
LIN {X 0,Y 242.168,Z 324.316,A -85,B 0,C 180,E1 -19365.141,E2 -19365.141} C_VEL
LIN {X 0,Y 242.074,Z 324.331,A -85,B 0,C 180,E1 -19368.624,E2 -19368.624} C_VEL
LIN {X 0,Y 242.014,Z 324.338,A -85,B 0,C 180,E1 -19372.18,E2 -19372.18} C_VEL
LIN {X 0,Y 242.067,Z 324.331,A -85,B 0,C 180,E1 -19375.838,E2 -19375.838} C_VEL
LIN {X 0,Y 242.031,Z 324.334,A -85,B 0,C 180,E1 -19379.58,E2 -19379.58} C_VEL
LIN {X 0,Y 241.99,Z 324.34,A -85,B 0,C 180,E1 -19383.491,E2 -19383.491} C_VEL
LIN {X 0,Y 241.999,Z 324.339,A -85,B 0,C 180,E1 -19387.58,E2 -19387.58} C_VEL
LIN {X 0,Y 241.944,Z 324.349,A -85,B 0,C 180,E1 -19391.921,E2 -19391.921} C_VEL
LIN {X 0,Y 241.935,Z 324.344,A -85,B 0,C 180,E1 -19396.572,E2 -19396.572} C_VEL
LIN {X 0,Y 241.958,Z 324.344,A -85,B 0,C 180,E1 -19400.281,E2 -19400.281} C_VEL
LIN {X 0,Y 242.022,Z 324.333,A -85,B 0,C 180,E1 -19404.495,E2 -19404.495} C_VEL
LIN {X 0,Y 241.977,Z 324.341,A -85,B 0,C 180,E1 -19408.48,E2 -19408.48} C_VEL
LIN {X 0,Y 242.01,Z 324.335,A -85,B 0,C 180,E1 -19412.313,E2 -19412.313} C_VEL
LIN {X 0,Y 242.043,Z 324.333,A -85,B 0,C 180,E1 -19416.015,E2 -19416.015} C_VEL
LIN {X 0,Y 242.024,Z 324.336,A -85,B 0,C 180,E1 -19419.607,E2 -19419.607} C_VEL
LIN {X 0,Y 242.13,Z 324.326,A -85,B 0,C 180,E1 -19423.307,E2 -19423.307} C_VEL
LIN {X 0,Y 242.171,Z 324.316,A -85,B 0,C 180,E1 -19428.279,E2 -19428.279} C_VEL
LIN {X 0,Y 242.397,Z 324.289,A -85,B 0,C 180,E1 -19431.665,E2 -19431.665} C_VEL
LIN {X 0,Y 242.255,Z 324.31,A -85,B 0,C 180,E1 -19435.007,E2 -19435.007} C_VEL
LIN {X 0,Y 242.638,Z 324.257,A -85,B 0,C 180,E1 -19438.34,E2 -19438.34} C_VEL
LIN {X 0,Y 242.635,Z 324.259,A -85,B 0,C 180,E1 -19441.66,E2 -19441.66} C_VEL
LIN {X 0,Y 242.408,Z 324.288,A -85,B 0,C 180,E1 -19446.66,E2 -19446.66} C_VEL
LIN {X 0,Y 242.27,Z 324.305,A -85,B 0,C 180,E1 -19450.024,E2 -19450.024} C_VEL
LIN {X 0,Y 242.142,Z 324.32,A -85,B 0,C 180,E1 -19455.143,E2 -19455.143} C_VEL
LIN {X 0,Y 242.053,Z 324.335,A -85,B 0,C 180,E1 -19458.626,E2 -19458.626} C_VEL
LIN {X 0,Y 242.006,Z 324.338,A -85,B 0,C 180,E1 -19462.181,E2 -19462.181} C_VEL
LIN {X 0,Y 242.035,Z 324.326,A -85,B 0,C 180,E1 -19465.821,E2 -19465.821} C_VEL
LIN {X 0,Y 241.973,Z 324.338,A -85,B 0,C 180,E1 -19469.588,E2 -19469.588} C_VEL
LIN {X 0,Y 241.99,Z 324.341,A -85,B 0,C 180,E1 -19473.491,E2 -19473.491} C_VEL
LIN {X 0,Y 241.999,Z 324.34,A -85,B 0,C 180,E1 -19477.581,E2 -19477.581} C_VEL
LIN {X 0,Y 242.041,Z 324.495,A -85,B 0,C 180,E1 -19480.204,E2 -19480.204} C_VEL
LIN {X 0,Y 242.855,Z 328.931,A -85,B 0,C 180,E1 -19483.991,E2 -19483.991} C_VEL
LIN {X 0,Y 243.181,Z 330.687,A -85,B 0,C 180,E1 -19485.444,E2 -19485.444} C_VEL
LIN {X 0,Y 242.826,Z 332.412,A -85,B 0,C 180,E1 -19486.772,E2 -19486.772} C_VEL
LIN {X 0,Y 240.511,Z 335.491,A -85,B 0,C 180,E1 -19488.938,E2 -19488.938} C_VEL
LIN {X 0,Y 237.734,Z 339.266,A -85,B 0,C 180,E1 -19491.593,E2 -19491.593} C_VEL
LIN {X 0,Y 237.474,Z 340.496,A -85,B 0,C 180,E1 -19492.507,E2 -19492.507} C_VEL
LIN {X 0,Y 237.052,Z 343.417,A -85,B 0,C 180,E1 -19494.681,E2 -19494.681} C_VEL
LIN {X 0,Y 235.492,Z 350.635,A -85,B 0,C 180,E1 -19499.937,E2 -19499.937} C_VEL
LIN {X 0,Y 234.777,Z 354.3,A -85,B 0,C 180,E1 -19502.567,E2 -19502.567} C_VEL
LIN {X 0,Y 236.588,Z 368.48,A -85,B 0,C 180,E1 -19503.61,E2 -19503.61} C_VEL
LIN {X 0,Y 237.947,Z 381.858,A -85,B 0,C 180,E1 -19504.928,E2 -19504.928} C_VEL
LIN {X 0,Y 238.79,Z 393.186,A -85,B 0,C 180,E1 -19506.33,E2 -19506.33} C_VEL
LIN {X 0,Y 239.279,Z 404.372,A -85,B 0,C 180,E1 -19508.007,E2 -19508.007} C_VEL
LIN {X 0,Y 239.183,Z 410.793,A -85,B 0,C 180,E1 -19509.128,E2 -19509.128} C_VEL
LIN {X 0,Y 237.292,Z 421.577,A -85,B 0,C 180,E1 -19511.286,E2 -19511.286} C_VEL
LIN {X 0,Y 235.8,Z 430.577,A -85,B 0,C 180,E1 -19513.552,E2 -19513.552} C_VEL
LIN {X 0,Y 234.56,Z 438.781,A -85,B 0,C 180,E1 -19516.131,E2 -19516.131} C_VEL
LIN {X 0,Y 233.724,Z 445.381,A -85,B 0,C 180,E1 -19518.729,E2 -19518.729} C_VEL
LIN {X 0,Y 233.304,Z 450.618,A -85,B 0,C 180,E1 -19521.337,E2 -19521.337} C_VEL
LIN {X 0,Y 233.249,Z 454.57,A -85,B 0,C 180,E1 -19523.892,E2 -19523.892} C_VEL
LIN {X 0,Y 233.214,Z 457.537,A -85,B 0,C 180,E1 -19526.545,E2 -19526.545} C_VEL
LIN {X 0,Y 233.371,Z 458.908,A -85,B 0,C 180,E1 -19528.274,E2 -19528.274} C_VEL
LIN {X 0,Y 233.596,Z 459.832,A -85,B 0,C 180,E1 -19530,E2 -19530} C_VEL
LIN {X 0,Y 233.097,Z 460.374,A -85,B 0,C 180,E1 -19533.457,E2 -19533.457} C_VEL
LIN {X 0,Y 232.955,Z 459.958,A -85,B 0,C 180,E1 -19535.388,E2 -19535.388} C_VEL
LIN {X 0,Y 233.093,Z 458.132,A -85,B 0,C 180,E1 -19538.671,E2 -19538.671} C_VEL
LIN {X 0,Y 233.412,Z 456.601,A -85,B 0,C 180,E1 -19540.408,E2 -19540.408} C_VEL
LIN {X 0,Y 234.199,Z 453.516,A -85,B 0,C 180,E1 -19543.007,E2 -19543.007} C_VEL
LIN {X 0,Y 235.642,Z 449.466,A -85,B 0,C 180,E1 -19545.571,E2 -19545.571} C_VEL
LIN {X 0,Y 237.507,Z 444.347,A -85,B 0,C 180,E1 -19548.102,E2 -19548.102} C_VEL
LIN {X 0,Y 240.082,Z 436.874,A -85,B 0,C 180,E1 -19551.014,E2 -19551.014} C_VEL
LIN {X 0,Y 243.115,Z 428.882,A -85,B 0,C 180,E1 -19553.421,E2 -19553.421} C_VEL
LIN {X 0,Y 246.573,Z 419.176,A -85,B 0,C 180,E1 -19555.764,E2 -19555.764} C_VEL
LIN {X 0,Y 248.217,Z 410.334,A -85,B 0,C 180,E1 -19557.677,E2 -19557.677} C_VEL
LIN {X 0,Y 249.087,Z 400.568,A -85,B 0,C 180,E1 -19559.588,E2 -19559.588} C_VEL
LIN {X 0,Y 249.054,Z 390.807,A -85,B 0,C 180,E1 -19561.393,E2 -19561.393} C_VEL
LIN {X 0,Y 248.143,Z 380.31,A -85,B 0,C 180,E1 -19563.246,E2 -19563.246} C_VEL
LIN {X 0,Y 246.19,Z 369.312,A -85,B 0,C 180,E1 -19565.197,E2 -19565.197} C_VEL
LIN {X 0,Y 242.873,Z 357.021,A -85,B 0,C 180,E1 -19567.451,E2 -19567.451} C_VEL
LIN {X 0,Y 241.553,Z 353.061,A -85,B 0,C 180,E1 -19568.226,E2 -19568.226} C_VEL
LIN {X 0,Y 239.282,Z 348.468,A -85,B 0,C 180,E1 -19569.344,E2 -19569.344} C_VEL
LIN {X 0,Y 238.815,Z 346.743,A -85,B 0,C 180,E1 -19569.646,E2 -19569.646} C_VEL
LIN {X 0,Y 238.394,Z 343.741,A -85,B 0,C 180,E1 -19572.692,E2 -19572.692} C_VEL
LIN {X 0,Y 237.66,Z 339.865,A -85,B 0,C 180,E1 -19577.144,E2 -19577.144} C_VEL
LIN {X 0,Y 237.079,Z 336.602,A -85,B 0,C 180,E1 -19581.499,E2 -19581.499} C_VEL
LIN {X 0,Y 236.625,Z 334.013,A -85,B 0,C 180,E1 -19585.645,E2 -19585.645} C_VEL
LIN {X 0,Y 236.252,Z 331.999,A -85,B 0,C 180,E1 -19589.621,E2 -19589.621} C_VEL
LIN {X 0,Y 236.037,Z 330.461,A -85,B 0,C 180,E1 -19593.472,E2 -19593.472} C_VEL
LIN {X 0,Y 235.774,Z 329.319,A -85,B 0,C 180,E1 -19597.527,E2 -19597.527} C_VEL
LIN {X 0,Y 235.708,Z 328.453,A -85,B 0,C 180,E1 -19602.652,E2 -19602.652} C_VEL
LIN {X 0,Y 235.69,Z 328.252,A -85,B 0,C 180,E1 -19606.199,E2 -19606.199} C_VEL
LIN {X 0,Y 235.928,Z 328.435,A -85,B 0,C 180,E1 -19611.434,E2 -19611.434} C_VEL
LIN {X 0,Y 236.08,Z 329.222,A -85,B 0,C 180,E1 -19616.586,E2 -19616.586} C_VEL
LIN {X 0,Y 236.257,Z 329.576,A -85,B 0,C 180,E1 -19617.656,E2 -19617.656} C_VEL
LIN {X 0,Y 237.479,Z 332.038,A -85,B 0,C 180,E1 -19618.357,E2 -19618.357} C_VEL
LIN {X 0,Y 239.985,Z 334.797,A -85,B 0,C 180,E1 -19619.518,E2 -19619.518} C_VEL
LIN {X 0,Y 241.926,Z 338.091,A -85,B 0,C 180,E1 -19620.52,E2 -19620.52} C_VEL
LIN {X 0,Y 242.599,Z 338.939,A -85,B 0,C 180,E1 -19620.83,E2 -19620.83} C_VEL
LIN {X 0,Y 248.286,Z 349.615,A -85,B 0,C 180,E1 -19623.856,E2 -19623.856} C_VEL
LIN {X 0,Y 250.93,Z 355.749,A -85,B 0,C 180,E1 -19625.475,E2 -19625.475} C_VEL
LIN {X 0,Y 253.518,Z 364.439,A -85,B 0,C 180,E1 -19627.542,E2 -19627.542} C_VEL
LIN {X 0,Y 255.011,Z 372.867,A -85,B 0,C 180,E1 -19629.518,E2 -19629.518} C_VEL
LIN {X 0,Y 255.196,Z 374.528,A -85,B 0,C 180,E1 -19629.911,E2 -19629.911} C_VEL
LIN {X 0,Y 252.545,Z 383.843,A -85,B 0,C 180,E1 -19631.562,E2 -19631.562} C_VEL
LIN {X 0,Y 249.682,Z 392.484,A -85,B 0,C 180,E1 -19633.428,E2 -19633.428} C_VEL
LIN {X 0,Y 246.45,Z 401.033,A -85,B 0,C 180,E1 -19635.72,E2 -19635.72} C_VEL
LIN {X 0,Y 243.764,Z 407.569,A -85,B 0,C 180,E1 -19637.929,E2 -19637.929} C_VEL
LIN {X 0,Y 240.733,Z 414.401,A -85,B 0,C 180,E1 -19640.897,E2 -19640.897} C_VEL
LIN {X 0,Y 238.297,Z 419.483,A -85,B 0,C 180,E1 -19643.896,E2 -19643.896} C_VEL
LIN {X 0,Y 236.401,Z 423.006,A -85,B 0,C 180,E1 -19646.889,E2 -19646.889} C_VEL
LIN {X 0,Y 234.961,Z 425.188,A -85,B 0,C 180,E1 -19649.838,E2 -19649.838} C_VEL
LIN {X 0,Y 233.988,Z 426.172,A -85,B 0,C 180,E1 -19652.753,E2 -19652.753} C_VEL
LIN {X 0,Y 233.394,Z 426.05,A -85,B 0,C 180,E1 -19655.606,E2 -19655.606} C_VEL
LIN {X 0,Y 233.132,Z 424.889,A -85,B 0,C 180,E1 -19658.39,E2 -19658.39} C_VEL
LIN {X 0,Y 233.273,Z 422.342,A -85,B 0,C 180,E1 -19661.514,E2 -19661.514} C_VEL
LIN {X 0,Y 233.622,Z 419.607,A -85,B 0,C 180,E1 -19663.781,E2 -19663.781} C_VEL
LIN {X 0,Y 234.21,Z 415.538,A -85,B 0,C 180,E1 -19666.356,E2 -19666.356} C_VEL
LIN {X 0,Y 235.106,Z 409.571,A -85,B 0,C 180,E1 -19669.257,E2 -19669.257} C_VEL
LIN {X 0,Y 236.41,Z 401.796,A -85,B 0,C 180,E1 -19672.173,E2 -19672.173} C_VEL
LIN {X 0,Y 237.842,Z 393.321,A -85,B 0,C 180,E1 -19674.695,E2 -19674.695} C_VEL
LIN {X 0,Y 239.564,Z 383.353,A -85,B 0,C 180,E1 -19677.052,E2 -19677.052} C_VEL
LIN {X 0,Y 241.34,Z 372.447,A -85,B 0,C 180,E1 -19679.12,E2 -19679.12} C_VEL
LIN {X 0,Y 242.983,Z 360.502,A -85,B 0,C 180,E1 -19680.903,E2 -19680.903} C_VEL
LIN {X 0,Y 243.171,Z 357.68,A -85,B 0,C 180,E1 -19681.282,E2 -19681.282} C_VEL
LIN {X 0,Y 240.789,Z 345.84,A -85,B 0,C 180,E1 -19682.867,E2 -19682.867} C_VEL
LIN {X 0,Y 237.483,Z 334.053,A -85,B 0,C 180,E1 -19684.223,E2 -19684.223} C_VEL
LIN {X 0,Y 234.735,Z 325.247,A -85,B 0,C 180,E1 -19685.124,E2 -19685.124} C_VEL
LIN {X 0,Y 234.925,Z 325.223,A -85,B 0,C 180,E1 -19688.962,E2 -19688.962} C_VEL
LIN {X 0,Y 235.056,Z 325.207,A -85,B 0,C 180,E1 -19693.092,E2 -19693.092} C_VEL
LIN {X 0,Y 235.11,Z 325.198,A -85,B 0,C 180,E1 -19697.922,E2 -19697.922} C_VEL
LIN {X 0,Y 235.321,Z 325.174,A -85,B 0,C 180,E1 -19701.412,E2 -19701.412} C_VEL
LIN {X 0,Y 235.358,Z 325.167,A -85,B 0,C 180,E1 -19703.14,E2 -19703.14} C_VEL
LIN {X 0,Y 235.596,Z 325.138,A -85,B 0,C 180,E1 -19708.291,E2 -19708.291} C_VEL
LIN {X 0,Y 235.596,Z 325.134,A -85,B 0,C 180,E1 -19711.709,E2 -19711.709} C_VEL
LIN {X 0,Y 235.358,Z 325.167,A -85,B 0,C 180,E1 -19716.86,E2 -19716.86} C_VEL
LIN {X 0,Y 235.215,Z 325.186,A -85,B 0,C 180,E1 -19720.328,E2 -19720.328} C_VEL
LIN {X 0,Y 235.115,Z 325.195,A -85,B 0,C 180,E1 -19725.606,E2 -19725.606} C_VEL
LIN {X 0,Y 235.01,Z 325.209,A -85,B 0,C 180,E1 -19729.206,E2 -19729.206} C_VEL
LIN {X 0,Y 234.962,Z 325.214,A -85,B 0,C 180,E1 -19732.883,E2 -19732.883} C_VEL
LIN {X 0,Y 234.971,Z 325.215,A -85,B 0,C 180,E1 -19736.657,E2 -19736.657} C_VEL
LIN {X 0,Y 234.933,Z 325.218,A -85,B 0,C 180,E1 -19740.568,E2 -19740.568} C_VEL
LIN {X 0,Y 234.961,Z 325.216,A -85,B 0,C 180,E1 -19744.633,E2 -19744.633} C_VEL
LIN {X 0,Y 234.943,Z 325.215,A -85,B 0,C 180,E1 -19748.945,E2 -19748.945} C_VEL
LIN {X 0,Y 234.888,Z 325.226,A -85,B 0,C 180,E1 -19753.486,E2 -19753.486} C_VEL
LIN {X 0,Y 234.888,Z 325.222,A -85,B 0,C 180,E1 -19756.514,E2 -19756.514} C_VEL
LIN {X 0,Y 234.92,Z 325.221,A -85,B 0,C 180,E1 -19761.079,E2 -19761.079} C_VEL
LIN {X 0,Y 234.952,Z 325.216,A -85,B 0,C 180,E1 -19765.366,E2 -19765.366} C_VEL
LIN {X 0,Y 234.934,Z 325.222,A -85,B 0,C 180,E1 -19769.433,E2 -19769.433} C_VEL
LIN {X 0,Y 234.996,Z 325.211,A -85,B 0,C 180,E1 -19773.794,E2 -19773.794} C_VEL
LIN {X 0,Y 234.993,Z 325.213,A -85,B 0,C 180,E1 -19778.968,E2 -19778.968} C_VEL
LIN {X 0,Y 235.066,Z 325.203,A -85,B 0,C 180,E1 -19783.086,E2 -19783.086} C_VEL
LIN {X 0,Y 235.103,Z 325.196,A -85,B 0,C 180,E1 -19787.922,E2 -19787.922} C_VEL
LIN {X 0,Y 235.329,Z 325.171,A -85,B 0,C 180,E1 -19791.413,E2 -19791.413} C_VEL
LIN {X 0,Y 235.371,Z 325.167,A -85,B 0,C 180,E1 -19793.141,E2 -19793.141} C_VEL
LIN {X 0,Y 235.597,Z 325.134,A -85,B 0,C 180,E1 -19798.291,E2 -19798.291} C_VEL
LIN {X 0,Y 235.594,Z 325.136,A -85,B 0,C 180,E1 -19801.71,E2 -19801.71} C_VEL
LIN {X 0,Y 235.36,Z 325.168,A -85,B 0,C 180,E1 -19806.86,E2 -19806.86} C_VEL
LIN {X 0,Y 235.217,Z 325.185,A -85,B 0,C 180,E1 -19810.328,E2 -19810.328} C_VEL
LIN {X 0,Y 235.089,Z 325.198,A -85,B 0,C 180,E1 -19815.608,E2 -19815.608} C_VEL
LIN {X 0,Y 234.993,Z 325.211,A -85,B 0,C 180,E1 -19819.207,E2 -19819.207} C_VEL
LIN {X 0,Y 234.949,Z 325.213,A -85,B 0,C 180,E1 -19822.884,E2 -19822.884} C_VEL
LIN {X 0,Y 234.949,Z 325.208,A -85,B 0,C 180,E1 -19826.66,E2 -19826.66} C_VEL
LIN {X 0,Y 234.902,Z 325.224,A -85,B 0,C 180,E1 -19830.572,E2 -19830.572} C_VEL
LIN {X 0,Y 234.962,Z 325.217,A -85,B 0,C 180,E1 -19834.633,E2 -19834.633} C_VEL
LIN {X 0,Y 234.952,Z 325.219,A -85,B 0,C 180,E1 -19839.467,E2 -19839.467} C_VEL
LIN {X 0,Y 235.018,Z 325.491,A -85,B 0,C 180,E1 -19840.011,E2 -19840.011} C_VEL
LIN {X 0,Y 235.927,Z 330.441,A -85,B 0,C 180,E1 -19844.362,E2 -19844.362} C_VEL
LIN {X 0,Y 236.7,Z 334.71,A -85,B 0,C 180,E1 -19847.927,E2 -19847.927} C_VEL
LIN {X 0,Y 237.491,Z 339.271,A -85,B 0,C 180,E1 -19851.578,E2 -19851.578} C_VEL
LIN {X 0,Y 237.474,Z 340.496,A -85,B 0,C 180,E1 -19852.507,E2 -19852.507} C_VEL
LIN {X 0,Y 236.713,Z 342.337,A -85,B 0,C 180,E1 -19853.843,E2 -19853.843} C_VEL
LIN {X 0,Y 234.863,Z 344.222,A -85,B 0,C 180,E1 -19855.134,E2 -19855.134} C_VEL
LIN {X 0,Y 230.287,Z 348.018,A -85,B 0,C 180,E1 -19857.716,E2 -19857.716} C_VEL
LIN {X 0,Y 228.751,Z 349.939,A -85,B 0,C 180,E1 -19859.086,E2 -19859.086} C_VEL
LIN {X 0,Y 228.509,Z 350.58,A -85,B 0,C 180,E1 -19859.558,E2 -19859.558} C_VEL
LIN {X 0,Y 227.839,Z 353.848,A -85,B 0,C 180,E1 -19861.991,E2 -19861.991} C_VEL
LIN {X 0,Y 229.583,Z 367.821,A -85,B 0,C 180,E1 -19863.041,E2 -19863.041} C_VEL
LIN {X 0,Y 230.952,Z 381.407,A -85,B 0,C 180,E1 -19864.425,E2 -19864.425} C_VEL
LIN {X 0,Y 231.823,Z 393.847,A -85,B 0,C 180,E1 -19866.02,E2 -19866.02} C_VEL
LIN {X 0,Y 232.288,Z 404.96,A -85,B 0,C 180,E1 -19867.778,E2 -19867.778} C_VEL
LIN {X 0,Y 232.084,Z 411.255,A -85,B 0,C 180,E1 -19868.924,E2 -19868.924} C_VEL
LIN {X 0,Y 230.458,Z 420.42,A -85,B 0,C 180,E1 -19870.824,E2 -19870.824} C_VEL
LIN {X 0,Y 228.912,Z 429.156,A -85,B 0,C 180,E1 -19873.042,E2 -19873.042} C_VEL
LIN {X 0,Y 227.645,Z 437.526,A -85,B 0,C 180,E1 -19875.701,E2 -19875.701} C_VEL
LIN {X 0,Y 226.705,Z 444.239,A -85,B 0,C 180,E1 -19878.375,E2 -19878.375} C_VEL
LIN {X 0,Y 226.251,Z 449.589,A -85,B 0,C 180,E1 -19881.065,E2 -19881.065} C_VEL
LIN {X 0,Y 226.182,Z 453.909,A -85,B 0,C 180,E1 -19883.892,E2 -19883.892} C_VEL
LIN {X 0,Y 226.148,Z 456.723,A -85,B 0,C 180,E1 -19886.437,E2 -19886.437} C_VEL
LIN {X 0,Y 226.286,Z 458.178,A -85,B 0,C 180,E1 -19888.22,E2 -19888.22} C_VEL
LIN {X 0,Y 226.538,Z 459.165,A -85,B 0,C 180,E1 -19890,E2 -19890} C_VEL
LIN {X 0,Y 226.022,Z 459.797,A -85,B 0,C 180,E1 -19893.566,E2 -19893.566} C_VEL
LIN {X 0,Y 225.884,Z 459.524,A -85,B 0,C 180,E1 -19895.356,E2 -19895.356} C_VEL
LIN {X 0,Y 225.888,Z 458.836,A -85,B 0,C 180,E1 -19897.149,E2 -19897.149} C_VEL
LIN {X 0,Y 226.37,Z 456.274,A -85,B 0,C 180,E1 -19900.736,E2 -19900.736} C_VEL
LIN {X 0,Y 227.265,Z 453.304,A -85,B 0,C 180,E1 -19903.411,E2 -19903.411} C_VEL
LIN {X 0,Y 228.774,Z 449.366,A -85,B 0,C 180,E1 -19906.051,E2 -19906.051} C_VEL
LIN {X 0,Y 230.766,Z 444.367,A -85,B 0,C 180,E1 -19908.65,E2 -19908.65} C_VEL
LIN {X 0,Y 233.48,Z 437.102,A -85,B 0,C 180,E1 -19911.638,E2 -19911.638} C_VEL
LIN {X 0,Y 236.654,Z 429.371,A -85,B 0,C 180,E1 -19914.101,E2 -19914.101} C_VEL
LIN {X 0,Y 240.218,Z 419.871,A -85,B 0,C 180,E1 -19916.498,E2 -19916.498} C_VEL
LIN {X 0,Y 242.229,Z 409.682,A -85,B 0,C 180,E1 -19918.803,E2 -19918.803} C_VEL
LIN {X 0,Y 243.161,Z 399.669,A -85,B 0,C 180,E1 -19920.865,E2 -19920.865} C_VEL
LIN {X 0,Y 243.025,Z 388.63,A -85,B 0,C 180,E1 -19923.002,E2 -19923.002} C_VEL
LIN {X 0,Y 241.834,Z 377.143,A -85,B 0,C 180,E1 -19925.179,E2 -19925.179} C_VEL
LIN {X 0,Y 239.52,Z 365.79,A -85,B 0,C 180,E1 -19927.382,E2 -19927.382} C_VEL
LIN {X 0,Y 236.944,Z 356.9,A -85,B 0,C 180,E1 -19929.24,E2 -19929.24} C_VEL
LIN {X 0,Y 235.148,Z 352.799,A -85,B 0,C 180,E1 -19930.264,E2 -19930.264} C_VEL
LIN {X 0,Y 234.658,Z 351.825,A -85,B 0,C 180,E1 -19930.536,E2 -19930.536} C_VEL
LIN {X 0,Y 232.429,Z 348.282,A -85,B 0,C 180,E1 -19931.725,E2 -19931.725} C_VEL
LIN {X 0,Y 231.538,Z 345.556,A -85,B 0,C 180,E1 -19932.37,E2 -19932.37} C_VEL
LIN {X 0,Y 230.787,Z 341.637,A -85,B 0,C 180,E1 -19936.959,E2 -19936.959} C_VEL
LIN {X 0,Y 230.377,Z 339.242,A -85,B 0,C 180,E1 -19940.16,E2 -19940.16} C_VEL
LIN {X 0,Y 229.843,Z 336.467,A -85,B 0,C 180,E1 -19944.481,E2 -19944.481} C_VEL
LIN {X 0,Y 229.445,Z 334.287,A -85,B 0,C 180,E1 -19948.619,E2 -19948.619} C_VEL
LIN {X 0,Y 229.182,Z 332.559,A -85,B 0,C 180,E1 -19952.787,E2 -19952.787} C_VEL
LIN {X 0,Y 228.929,Z 331.282,A -85,B 0,C 180,E1 -19957.072,E2 -19957.072} C_VEL
LIN {X 0,Y 228.828,Z 330.34,A -85,B 0,C 180,E1 -19962.197,E2 -19962.197} C_VEL
LIN {X 0,Y 228.822,Z 330.066,A -85,B 0,C 180,E1 -19965.776,E2 -19965.776} C_VEL
LIN {X 0,Y 229.017,Z 330.172,A -85,B 0,C 180,E1 -19971.174,E2 -19971.174} C_VEL
LIN {X 0,Y 229.069,Z 330.725,A -85,B 0,C 180,E1 -19974.829,E2 -19974.829} C_VEL
LIN {X 0,Y 230.284,Z 333.284,A -85,B 0,C 180,E1 -19975.679,E2 -19975.679} C_VEL
LIN {X 0,Y 233.16,Z 336.086,A -85,B 0,C 180,E1 -19977.191,E2 -19977.191} C_VEL
